// TwinCAT 3 PLC project IBF_Devices
// Title: IBF_Devices
// Company: Industrial Brains B.V.
// ProjectVersion: 0.0.0.0
// ProgramVersion: 3.1.4023.0
// CompilerDefines: InclSerialCom := 'true'
// libraries:
//   IBF_Utilities, * (Industrial Brains B.V.)
//   Tc2_Drive, * (Beckhoff Automation GmbH)
//   Tc2_EtherCAT, * (Beckhoff Automation GmbH)
//   Tc2_IoFunctions, * (Beckhoff Automation GmbH)
//   Tc2_Math, * (Beckhoff Automation GmbH)
//   Tc2_MC2, * (Beckhoff Automation GmbH)
//   Tc2_MC2_Drive, * (Beckhoff Automation GmbH)
//   Tc2_Standard, * (Beckhoff Automation GmbH)
//   Tc2_System, * (Beckhoff Automation GmbH)
//   Tc2_Utilities, * (Beckhoff Automation GmbH)
//   Tc3_Module, * (Beckhoff Automation GmbH)
//   VisuDialogs, * (System)
// project tree:
//   Axis/FunctionBlocks/Servo/ Fb_DevAxisDelta.TcPOU, Fb_DevAxis.TcPOU
//   / GlobalTextList.TcGTLO, PlcTask.TcTTO, Visualization Manager.TcVMO (not stored), VISU_TASK.TcTTO
//   GroupHandlers/ManualControlHandler/DataTypes/ UDT_DeviceID.TcDUT, UDT_HMI_ManualControl.TcDUT
//   GroupHandlers/ManualControlHandler/HMI/DeviceScreens/ VisuAnalogAxisControl.TcVIS, VisuAnalogOutControl.TcVIS, VisuAnlogInputControl.TcVIS, VisuAxisControl.TcVIS, VisuCylinderControl.TcVIS, VisuDigitalInputControl.TcVIS, VisuDigitalOutControl.TcVIS, VisuDoublePWMControl.TcVIS, VisuEncoderInput.TcVIS, VisuKL15XXControl.TcVIS, VisuKL5151Control.TcVIS, VisuPushbuttonLightControl.TcVIS, VisuPWMControl.TcVIS, VisuTwoVelocityAxisControl.TcVIS, VisuUndefinedControl.TcVIS, VisuValveControl.TcVIS
//   GroupHandlers/ManualControlHandler/HMI/ ManualControl.TcVIS
//   GVL/ GVL_Devices.TcGVL
//   _TESTS/ PRG_TEST_FB_DEVAXIS.TcPOU, PRG_TEST_FB_DEVVALVE.TcPOU, PRG_TEST_FB_MANUALCONTROLLER.TcPOU, PRG_TEST_GLOBAL.TcPOU, VISU_TEST.TcVIS, VISU_TEST_LOGIN.TcVIS
//   Actuators/Cylinder/DataTypes/ E_CylinderCmd.TcTLEO (not stored), E_ValveResetState.TcTLEO (not stored)
//   Actuators/Cylinder/DataTypes/ManualControls/ UDT_ManualValveControl.TcDUT (not stored)
//   Actuators/Cylinder/Functions/ Fb_DevCylWithFbk.TcPOU, FB_DevValve.TcPOU
//   Axis/DataTypes/ E_AxisCmd.TcTLEO (not stored), UDT_AxisData.TcDUT (not stored), UDT_AxVal.TcDUT (not stored), UDT_ManualAxisCtrl.TcDUT (not stored)
//   Axis/FunctionBlocks/Analog/ FB_DevAnalogAxis.TcPOU, ST_ManualAnalogAxisCtrl.TcDUT (not stored)
//   Axis/FunctionBlocks/ServoHybrid/ FB_DevBasicACAxis.TcPOU, FB_DevHybridAc.TcPOU
//   Axis/FunctionBlocks/TwoVelocityControl/DataTypes/ st_ManualDigitalMotorControl.TcDUT
//   Axis/FunctionBlocks/TwoVelocityControl/ FB_DevTwoVelocityAxis.TcPOU
//   Axis/Interface/ iTwoDirectionalMotor.TcIO, iTwoDirectionalMotorWithFast.TcIO (not stored)
//   BaseFunctions/ FB_DevBase.TcPOU, UDT_DevManualCtrl.TcDUT (not stored)
//   Buttons/Functions/ FB_DevHMIButton.TcPOU, FB_DevPushbuttonLight.TcPOU, FB_DevPushButton.TcPOU
//   CounterCards/FunctionBlocks/KL1512/ FB_DevKL1512.TcPOU (not stored)
//   CounterCards/FunctionBlocks/KL5151/ FB_DevKL5151.TcPOU
//   CounterCards/Interfaces/ iCounter.TcIO (not stored)
//   CounterCards/ st_ManualCounterControl.TcDUT (not stored)
//   DevTypes/ E_Devices.TcTLEO
//   Encoders/FunctionBlocks/ FB_EncoderBase.TcPOU, FB_EncoderInput.TcPOU
//   GroupHandlers/ManualControlHandler/ FB_ManualController.TcPOU
//   HardwareDiagnostics/ FB_ELModuleDiag.TcPOU (not stored)
//   Heaters/ FB_DevDoublePWM.TcPOU, FB_DevPWMGenerator.TcPOU
//   Lights/Functions/ Fb_DevLight.TcPOU
//   Outputs/AnalogOutputs/ FB_DevAnalogOutput.TcPOU, FB_DevAnalogOutputScaled.TcPOU
//   Outputs/DigitalOutputs/ FB_DevDigitalOutput.TcPOU
//   Sensors/AnalogInput/FunctionBlocks/ FB_DevAnalogInput.TcPOU, FB_DevAnalogInputScaled.TcPOU, FB_DevHDAnalogInAutoCalibrate.TcPOU, FB_DevAnalogInAutoCalibrate.TcPOU, FB_DevHDAnalogInputScaled.TcPOU, FB_DevHDAnalogInput.TcPOU
//   Sensors/DigitalSensor/FunctionBlocks/ Fb_DevDigitalInput.TcPOU, Fb_DevDigitalInputFunctions.TcPOU
//   Sensors/FootPedals/DataTypes/ E_FootpedalPos.TcTLEO (not stored)
//   Sensors/FootPedals/FunctionBlocks/ FB_EfkaEB301A_FootPedal.TcPOU
//   Sensors/ModuleSpecific/EL3556_Loadcell/ Fb_DevEL3356_LoadCell.TcPOU (not stored)
//   Version/ Global_Version.TcGVL
// real-time tasks:
//   TASK PlcTask: cycle T#10ms, priority 10, ADS port 350
//   TASK VISU_TASK: cycle T#200000us, priority 12, ADS port 351
// motion (NC):
//   TASK NC-Task 1 SAF: cycle T#2ms, priority 4, ADS port 501
//   TASK NC-Task 1 SVB: cycle T#10ms, priority 8, ADS port 511
//   AXIS Axis 1 (id 1)
//     OtherSettings: AllowMotionCmdToSlave=true
//     encoder EncType=1
//       SoftEndMinControl: Enable=true
//       SoftEndMaxControl: Enable=true, Range=1000
//     drive DrvType=5
//       Analog: TorqueSetpointScale=10, ScaleFactorActTorque=0.1
//       TimeComp: TaskDelayCycles=1
//     controller CtrType=1
//       CtrPara: PriorControlFactor=1
//         Observer: BandWidth=20
// variable links:
//   IBF_Devices Instance <-> NC-Task 1 SAF/Axes/Axis 1
//     PlcTask Inputs/PRG_TEST_FB_DEVAXIS.fbDevAxis.AxisRef.NcToPlc <-> Outputs/ToPlc
//     PlcTask Outputs/PRG_TEST_FB_DEVAXIS.fbDevAxis.AxisRef.PlcToNc <-> Inputs/FromPlc

CONFIGURATION IBF_Devices
    RESOURCE PLC ON TwinCAT3
        TASK PlcTask(INTERVAL := T#10ms, PRIORITY := 10);
        TASK VISU_TASK(INTERVAL := T#200000us, PRIORITY := 12);
        PROGRAM PRG_TEST_GLOBAL WITH PlcTask : PRG_TEST_GLOBAL;
        PROGRAM PRG_TEST_FB_DEVAXIS WITH PlcTask : PRG_TEST_FB_DEVAXIS;
        PROGRAM PRG_TEST_FB_DEVVALVE WITH PlcTask : PRG_TEST_FB_DEVVALVE;
        PROGRAM PRG_TEST_FB_MANUALCONTROLLER WITH PlcTask : PRG_TEST_FB_MANUALCONTROLLER;
        PROGRAM VisuElems_Visu_Prg WITH VISU_TASK : VisuElems.Visu_Prg;
    END_RESOURCE
END_CONFIGURATION

// ---- GroupHandlers/ManualControlHandler/DataTypes/UDT_DeviceID.TcDUT
TYPE UDT_DeviceID :
STRUCT
	sName			: STRING	; // device name
	sType			: STRING	; // Type of device [string for visu]
	pFunction		: POINTER TO FB_DevBase ; // Pointer to the device
END_STRUCT
END_TYPE

// ---- GroupHandlers/ManualControlHandler/DataTypes/UDT_HMI_ManualControl.TcDUT
TYPE UDT_HMI_ManualControl : // The link between HMI and FB
STRUCT
	refSelectedDevice	: REFERENCE TO FB_DevBase; // Reference to currently selected device
	nSelectedDevice		: UDINT; // Combo box index
	bReset 				: BOOL;
	bEnabled			: BOOL;	
	bBlocked			: BOOL;

	// References to all supported device types
	pDevValve			: POINTER TO FB_DevValve;
	pDevCylinder		: POINTER TO Fb_DevCylWithFbk; 
	pDevAxis			: POINTER TO Fb_DevAxis; 
	pDevPBL				: POINTER TO FB_DevPushbuttonLight;
	pDevDigitalInput	: POINTER TO Fb_DevDigitalInputFunctions;
	pDevAnalogInput		: POINTER TO FB_DevAnalogInput;
	pDevAnalogOut		: POINTER TO FB_DevAnalogOutput;
	pDevDigitalOut		: POINTER TO FB_DevDigitalOutput;
	pDevPWMController	: POINTER TO FB_DevPWMGenerator;
	pDevDoublePWM		: POINTER TO FB_DevDoublePWM;
	pDevEncoder			: POINTER TO FB_EncoderBase;
	pDevAnalogAxis		: POINTER TO FB_DevAnalogAxis;
	pDevTwoVelocityAxis	: POINTER TO FB_DevTwoVelocityAxis;
	pDevKL5151			: POINTER TO FB_DevKL5151;
	pDevKL1512			: POINTER TO FB_DevKL1512;
END_STRUCT
END_TYPE

// ---- Axis/FunctionBlocks/TwoVelocityControl/DataTypes/st_ManualDigitalMotorControl.TcDUT
TYPE st_ManualDigitalMotorControl : // commands from manual controller
STRUCT
	bManRunCW 		: BOOL ;
	bManRunCWFast	: BOOL ;
	bManRunCCw		: BOOL ;
	bManRunCCWFast	: BOOL ; 
END_STRUCT
END_TYPE

// ---- DevTypes/E_Devices.TcTLEO
{attribute 'qualified_only'}
{attribute 'strict'}
{attribute 'to_string'}
TYPE E_Devices :
(
	Undefined,
	Valve,
	Cylinder,
	Axis,
	PushButtonLight,
	DigitalSensor,
	AnalogSensor,
	DigitalOut,
	AnalogOut,
	PWMController,
	DoublePWMController,
	Encoder,
	AnalogAxis,
	TwoVelocityAxis,
	KL5151,
	KL1512
)INT;
END_TYPE

// ---- GVL/GVL_Devices.TcGVL
{attribute 'qualified_only'}
VAR_GLOBAL
	fbManualController : FB_ManualController;
END_VAR

// ---- Version/Global_Version.TcGVL
{attribute 'TcGenerated'}
{attribute 'no-analysis'}
{attribute 'linkalways'}
// This function has been automatically generated from the project information.
VAR_GLOBAL CONSTANT
	{attribute 'const_non_replaced'}
	stLibVersion_IBF_Devices : ST_LibVersion := (iMajor := 0, iMinor := 0, iBuild := 0, iRevision := 0, nFlags := 0, sVersion := '0.0.0.0');
END_VAR

// ---- Axis/Interface/iTwoDirectionalMotor.TcIO
INTERFACE iTwoDirectionalMotor // Two directional motor control

METHOD CmdRunCCW : BOOL
VAR_INPUT
END_VAR
END_METHOD

METHOD CmdRunCW : BOOL
VAR_INPUT
END_VAR
END_METHOD

METHOD Init : BOOL
VAR_INPUT
	// Message location data
	nId				: UINT ; // Identification number of object
	nParentId		: UDINT ; // Id of higher level If aplicable (0 = no parent)
END_VAR
END_METHOD

END_INTERFACE

// ---- _TESTS/PRG_TEST_GLOBAL.TcPOU
PROGRAM INTERNAL PRG_TEST_GLOBAL // A place to call global function blocks (singletons) that can be used by all tests

Sys_Variables.fbSystemVariables();
GVL_Utilities.fbFaultHandler();

END_PROGRAM

// ---- _TESTS/PRG_TEST_FB_DEVAXIS.TcPOU
PROGRAM INTERNAL PRG_TEST_FB_DEVAXIS
VAR
	bEnableTests : BOOL;
	
	fbDevAxis : Fb_DevAxis;
	
	// Setpoints
	fVelocity : LREAL := 100;
	fPosition : LREAL := 500; // NOTE: software limit switch is at 1000 (/Axes/Axis 1/Enc/ Parameters)

	// Public commands
	bInit : BOOL;
	bCmdHalt : BOOL;
	bCmdHold : BOOL;
	bCmdHome : BOOL;
	bCmdReset : BOOL;
	bCmdMoveAbs : BOOL;
END_VAR

IF bEnableTests THEN
	fbDevAxis();
	
	IF bInit THEN
		bInit R= fbDevAxis.Init(
			nId					:= 1, 
			nParentId			:= 0, 
			bIcfCmdVelocityRpm	:= FALSE, 
			bIcfEnableForward	:= TRUE, 
			bIcfEnableReverse	:= TRUE, 
			bIcfAlwaysEnable	:= FALSE, 
			bIcfModuloAxis		:= FALSE, 
			bIcfSTOPresent		:= TRUE, 
			bIcfNCHomeSensor	:= FALSE, 
			mcHomingMode		:= MC_HomingMode.MC_DefaultHoming, 
			fSafeOverride		:= 20, 
			nEncTurnoverVal		:= 0,
			tEnableDelay		:= T#0S, 
			tDisabledelay		:= T#200MS
		);
	END_IF
		
	// Trigger commands
	IF bCmdHalt THEN bCmdHalt R= fbDevAxis.CmdHalt(fDeceleration := 1000, MC_BufferMode.MC_Aborting); END_IF
	IF bCmdHold THEN bCmdHold R= fbDevAxis.CmdHold(); END_IF
	IF bCmdHome THEN bCmdHome R= fbDevAxis.CmdHome(); END_IF
	IF bCmdReset THEN bCmdReset R= fbDevAxis.CmdReset(); END_IF
	IF bCmdMoveAbs THEN bCmdMoveAbs R= fbDevAxis.CmdMoveAbs(fPosition := fPosition, fVelocity := fVelocity, MC_BufferMode.MC_Aborting); END_IF
END_IF

END_PROGRAM

// ---- Axis/FunctionBlocks/Servo/Fb_DevAxis.TcPOU
{attribute 'reflection'}
FUNCTION_BLOCK PUBLIC Fb_DevAxis EXTENDS FB_DevBase
VAR_INPUT
	// ===== General Function input =====
		fCmdAcc			: LREAL := 15000;
		fCmdDec			: LREAL := 15000; 
	// ===== Master Axis =====
		refMasterAxis	: REFERENCE TO AXIS_REF ; // Master axis reference (if applicable)
		bReverseSlave	: BOOL 	:= FALSE; // Reverse slave axis relative to master
		fCmdGearRatio	: LREAL := 1 ; // Gear ratio Master/Slave (1/Ratio) 
	// Manual control reference
		stManualCtrl	: UDT_ManualAxisCtrl ;
END_VAR
VAR_OUTPUT
	// ====== State indications =======
		bHomed			: BOOL 	:= FALSE; 
		bError 			: BOOL 	:= FALSE;
		bStopped		: BOOL 	:= FALSE;
		bResetDone		: BOOL 	:= FALSE;
		bGearedAsSlave	: BOOL 	:= FALSE;
		bVelocityLimited: BOOL 	:= FALSE;  
		bIdle			: BOOL 	:= FALSE;
		fVelocity		: LREAL	:= 0	; // Axis velocity [rpm or units/sec] depending on config
		fActPosition	: LREAL := 0	; // Axis actual position [Units] depending on config	
		bReInTargetPos	: BOOL 	:= false; // rising edge axis is in position
	// ====== axis reference ======
		AxisRef			: AXIS_REF	; // Axis reference to hardware 
	// ====== Axis Settings ======
		fMaxVelo		: LREAL := 0 ; // Axis Maximum velocity
		fMaxAcc			: LREAL := 0 ; // Axis Maximum cceleration
		fMaxDec			: LREAL := 0 ; // axis Maxium deceleration 
	
//		fSafeVeloLimit	: LREAL	:= 200; // Safe velocity limit 
		tEnableDelay	: TIME 	:= T#0MS	;
		tDisableDelay	: TIME 	:= T#500MS  ;
	// ==== Axis data ====
		fEncoderTurnoverValue	: LREAL ;   
		
END_VAR
VAR // Axis configuration 
	// ===== HW Config Bits =====
		bIcfCmdVelocityRpm	: BOOL ; // input speeds in Rpm
		bIcfEnableForward 	: BOOL ; // Enable forward motion
 		bIcfEnableReverse	: BOOL ; // Enable reverse motion
		bIcfAlwaysEnable	: BOOL ; // 1 = Axis always enabled, 0 = Axis disabled at Idle 
		bIcfModuloAxis		: BOOL := FALSE ; // Show axis position as modulo
		bIcfSTOPresent		: BOOL := FALSE ; // Axis Safe torque off is present
		bIcfNCHomeSensor	: BOOL := FALSE ; // Homing sensor is inverted (NC)	
	// Command Modes
		mcHomingMode 		: MC_HomingMode := MC_direct ; // Homing Mode ( MC_DefaultHoming, MC_Direct, MC_ForceCallibration, MC_ResetCallibration)
	// Values from system
		McReadSysVelo		: MC_ReadParameter		; // Read Acceleration parameter from drive 
		McReadSysAcc		: MC_ReadParameter		; // Read Acceleration parameter from drive 
		McReadSysDec		: MC_ReadParameter		; // Read Acceleration parameter from drive 
END_VAR
VAR	// ====== Axis enable =====
		bCmdEnableAxis 		: BOOL 	:= FALSE; // Command to enable the axis (External)
		bInternalEnable		: BOOL 	:= FALSE; // internal enable command (turns off after set time, and on at new motion command
		bAxisIsEnabled		: BOOL 	:= false; // Axis is enabled and ready for commands
		bDelayedEnable		: BOOL 	:= false; // Delayed enable signal for motion commands
		TonMotionEnable		: TON 			; // Timer on for motion command enable
		TofIntAxisEnable	: TOF  			; // Timer off for internal axis enable 
		bSTOOK				: BOOL 	:= FALSE; // Axis safet torque off is ok
		tonSTOOK			: TON	; // Safe torque off ok timer
	// Parameter read status 
		Cmd_EnDriveParRead	: BOOL 			; // Enable parameter read 
	// ===== Physical Homing signal =====
		IAxisHome 	AT %I* 	: BOOL 			; // Axis homing sensor from PLC (if MC_DefaultHoming is used)
		IAxisSTOOK	AT %I* 	: BOOL 			; // Axis STO is ok
END_VAR
VAR	// =============== Motion status functions ================
	// =============== Motion function blocks =================
		fbMcPower 			: MC_Power		;		// FB for enable and override
		fbMcReset 			: MC_Reset		;		// FB to reset axis
		fbSoeReset			: FB_SoEReset	; 		// FB to reset axis hardware
		fbMcHome			: MC_Home		;		// Fb to home Axis
		fbHomeResetCalibrationFlag:MC_Home;			// Fb to clear calibration (homed) bit
		bResetCalibrationFlag : BOOL := FALSE; // When TRUE, the calibration bit (homing OK) will be reset. Set to TRUE on homing faults.
		fbMcStop 			: MC_Stop		;		// FB to stop axis
		fbMcHalt			: MC_Halt		;		// FB to halt axis
		fbMcJog				: MC_Jog		;		// FB to Jog axis
		fbMcMoveVelocity	: MC_MoveVelocity;		// FB to move with specified velocity until Next command is given
		fbMcGearInSlave		: MC_GearIn		;		// FB to gear axis to master 
		fbMcGearInDyn		: MC_GearInDyn	;		// FB to gear axis dynamicly to master
		fbMcGearOutSlave	: MC_GearOut	;		// FB to decouple gearing
		fbMcSetPosition		: MC_SetPosition;		// FB to Set axis position
//		fbMcWriteParameter	: MC_WriteParameterPersistent ; // FB to write parameters in persistend data

	(* PtoP Motion move commands are in arrays so multiple commands can be stacked *) 
		fbMCMoveRelative	: ARRAY [0..1] OF MC_MoveRelative	;		// FB to move relative
		fbMcMoveAbsolute	: ARRAY [0..1] OF MC_MoveAbsolute	;		// FB to move axis (velocity movement)
		fbMcMoveModulo		: ARRAY [0..1] OF MC_MoveModulo		;		// FB to move axis to modulo position
	// ===== Safe commands =====
		bCmdSafeStop		: BOOL ;
		bCmdSafeSpeed		: BOOL ; 
	// ===== Function execute triggers =====
		bExec_Reset					: BOOL := FALSE; // Execute reset
		bExec_Halt					: BOOL := FALSE; // Execute hold
		bExec_Home					: BOOL := FALSE; // Execute Home
		bExec_JogPositive			: BOOL := FALSE; // Execute Jog in positive direction
		bExec_JogNegative			: BOOL := FALSE; // Execute Jog in negative direction
		bExec_MoveVelocity			: BOOL := FALSE; // Execute move velocity
		bExec_MoveVelocityDynamic	: BOOL := FALSE; // Execute move velocity
		bExec_GearAsSlave			: BOOL := FALSE; // Execute gear as slave
		bExec_GearSlaveDyn			: BOOL := FALSE; // Execute gear slave dynamic
		bExec_GearOutSlave			: BOOL := FALSE; // Execute gear out slave
		bExec_SetPosition			: BOOL := FALSE; // execute set position
		
	(* PtoP Motion move commands are in arrays so multiple commands can be stacked *) 
		arExec_MoveRelative	: ARRAY [0..1] OF BOOL ; // Execute move relative
		arExec_MoveAbs		: ARRAY [0..1] OF BOOL ; // Execute move absolute reverse
		arExec_MoveModulo	: ARRAY [0..1] OF BOOL ; // Execute move modulo

		tonResetDone		: TON := (PT := T#300MS) ;

	// ===== Move ristrictions ======
		bCmdLimitVelocity 	: BOOL := FALSE			; // velocity limiting is active 
		fCmdVelocityLimit	: LREAL:= 100			; // Maximum velocity limit when velocity limiting is active  
		fSafeOverride		: LREAL:= 10 			; // [%] Safe velocity override  
		
	// ===== Internal variables =======
		fAcceleration		: LREAL := 0 ; // Acceleration used for functions 
		fDeceleration		: LREAL := 0 ; // Deceleration used for functions
		fLastCommandPosition: LREAL := 0 ; // Last given position command
		fLastCommandVelocity: LREAL := 0 ; // Last given Velocity command

	// Register command changes to make sure CmdMoveAbs is triggered
	{warning 'TODO: this is a workaround for a generic software design issue of DevAxis (needs state machine)'}
	bResetCmdMoveAbs : BOOL := TRUE;
		
END_VAR
VAR
	// ===== Loop variables =====
		i : DINT := 0 ; // For loop increment
	// ===== check variable ======
		rtrigInPosition	: R_TRIG ; // in position trigger
	// ===== Par write timer ===== 
END_VAR
VAR // Parameters 
	ParHomeOffset		: Udt_Parameter := (fValue := 0, fFactory := 0, bTeachable := FALSE)	; // Home position offset
END_VAR

// Call base function
SUPER^();

// ==== Check if axis is initiated =====
IF NOT bInitOk THEN 
	RETURN ; 
END_IF
// ===== Execute safe functions =====
	ExecSafeFunctions(); 
	
// ==== Execute organizational functions =====
	CallOrganizationFunctions();
// ==== execute motion functions =====
	CallMotionFunctions();

// ==== reset calibration ("homed") flag =====
fbHomeResetCalibrationFlag(
  Execute:=bResetCalibrationFlag,
  HomingMode:=MC_ResetCalibration,
  Axis:=AxisRef
);
bResetCalibrationFlag R= fbHomeResetCalibrationFlag.Done;


IF bHomed AND (NOT AxisRef.NcToPlc.StateDWord.1) // Check if drive is still homed
THEN 
	{warning 'TODO: Skip homing check if the drive is not connected (e.g., during automated tests of an axis with disabled hardware)'}
	bHomed := FALSE;
	IF NOT bManual THEN // Ignore homing error when in manual mode
		bError					:= TRUE							;
		stFault.Active 			:= TRUE 						;
		stFault.Description		:= 'Axis no longer homed';
		stFault.FaultType		:= E_FaultTypes.FF				;	
	END_IF
END_IF

METHOD PRIVATE CallMotionFunctions : BOOL
VAR_INPUT
END_VAR
// ===== block all other commands if axis is coupled =====
	IF NOT AxisRef.Status.Coupled THEN 
	// ===== Homing functions =====
		ExecHome		(); 
	
	// ===== Motion standstil commands =====
		ExecHalt		();
	
	// ===== Motion move functions
		ExecJog			();
		ExecMoveAbsolute();
		ExecMoveRelative();
		ExecMoveModulo	();
		ExecMoveVelocity();
	END_IF
	
// ===== Execute gearing functions =====
 IF __ISVALIDREF (refMasterAxis) THEN 
	ExecGearOut		();
	ExecGearIn		();
	ExecGearDynamic	();
 END_IF
	
// ====== reset velocity lmiting =====
	bVelocityLimited	:= bCmdLimitVelocity ;	
	bCmdLimitVelocity 	:= FALSE ; 

// ====== Reset acceleration deceleration values ======
	fAcceleration	:= fCmdAcc;
	fDeceleration	:= fCmdDec;
END_METHOD

METHOD PRIVATE CallOrganizationFunctions : BOOL
VAR_INPUT
END_VAR
// ==== execute organizational functions =====
	ExecReadStatus		(); 
	ExecEnable			();
	ExecReset			();
//	ExecWriteParameter	();
	ExecSetPosition		();
END_METHOD

METHOD PUBLIC CmdGearDynamic : BOOL // Set axis to geared, activates with variable gear ratio until geared out or stopped (if method is no longer called then gear ratio is locked to last value)
VAR_INPUT
	fGearRatio	:	LREAL	:= 1	; // Slave Axis gearing ratio (Master = 1/ fGearRatio = Slave)	
END_VAR
// check if master is present
	IF NOT __ISVALIDREF (refMasterAxis) THEN 
		bError					:= TRUE							;
		stFault.Active 			:= TRUE 						;
		stFault.Description		:= CONCAT('Axis master not found ', UDINT_TO_STRING(fbMcHalt.ErrorID));
		stFault.FaultType		:= E_FaultTypes.FF				;
	END_IF

// check if error is active
	IF bError THEN
		stFault.Active 			:= TRUE 						;
		stFault.Description		:= 'Call to CmdGearDynamic while axis has an error';
		stFault.FaultType		:= E_FaultTypes.CF				;	
		RETURN;
	END_IF

// set blocked command if halt is active 
	bBlockedCommand 		:= fbMcHalt.Active ;


// check if command buffer is empty 
	IF AxisRef.Status.CmdBuffered THEN 
		RETURN ;
	END_IF 

// Set command to true 
	bExec_GearSlaveDyn 	:= TRUE ;
	bInternalEnable		:= TRUE ;

// copy parameters
	fCmdGearRatio 		:= fGearRatio ;

// Reset CmdMoveAbs
bResetCmdMoveAbs := TRUE;

// Set feedback output 
	CmdGearDynamic 		:= bGearedAsSlave ;
END_METHOD

METHOD PUBLIC CmdGearIn : BOOL // Set axis to geared, activates with constant gear ratio until geared out or stopped
VAR_INPUT
	fGearRatio	:	LREAL	:= 1	; // Slave Axis gearing ratio (Master = 1/ fGearRatio = Slave)	
END_VAR
// Check if master is present
	IF NOT __ISVALIDREF (refMasterAxis) THEN 
		bError					:= TRUE							;
		stFault.Active 			:= TRUE 						;
		stFault.Description		:= CONCAT('Axis master not found ', UDINT_TO_STRING(fbMcHalt.ErrorID));
		stFault.FaultType		:= E_FaultTypes.FF				;
	END_IF

// check if error is active
	IF bError THEN
		stFault.Active 			:= TRUE 						;
		stFault.Description		:= 'Call to CmdGearIn while axis has an error';
		stFault.FaultType		:= E_FaultTypes.CF				;	
		RETURN;
	END_IF

// set blocked command if halt is active 
	bBlockedCommand := fbMcHalt.Active ;

// check if command buffer is empty 
	IF AxisRef.Status.CmdBuffered THEN 
		RETURN ;
	END_IF 
	
// Set command to true 
	bExec_GearAsSlave 	:= TRUE ;
	bInternalEnable		:= TRUE ;

// copy parameters
	fCmdGearRatio 				:= fGearRatio ;

// Reset CmdMoveAbs
bResetCmdMoveAbs := TRUE;

// Set feedback output 
	CmdGearIn := bGearedAsSlave ;
END_METHOD

METHOD CmdGearOut : BOOL
VAR_INPUT
END_VAR
// Check if master is present
	IF NOT __ISVALIDREF (refMasterAxis) THEN 
		bError					:= TRUE							;
		stFault.Active 			:= TRUE 						;
		stFault.Description		:= CONCAT('Axis master not found ', UDINT_TO_STRING(fbMcHalt.ErrorID));
		stFault.FaultType		:= E_FaultTypes.FF				;
	END_IF

// check if error is active
	IF bError THEN
		stFault.Active 			:= TRUE 						;
		stFault.Description		:= 'Call to CmdGearOut while axis has an error';
		stFault.FaultType		:= E_FaultTypes.CF				;	
		RETURN;
	END_IF

// set blocked command if halt is active 
bBlockedCommand := fbMcHalt.Active ;

// Set command to true
bExec_GearOutSlave 	:= TRUE ;
bExec_GearAsSlave	:= FALSE;
bExec_GearSlaveDyn 	:= FALSE;

// Reset CmdMoveAbs
bResetCmdMoveAbs := TRUE;

// Set feedback Output
CmdGearOut := fbMcGearOutSlave.Done;
END_METHOD

METHOD PUBLIC CmdHalt : BOOL
VAR_INPUT
	fDeceleration 	: LREAL := 0 ; // command deceleration
	mcBuffermode	: MC_BufferMode ; // Buffermode defines how the previous command is executed.
END_VAR
// Set command to true 
bExec_Halt 		:= TRUE ;
bInternalEnable	:= TRUE ;

// copy parameters
fbMcHalt.Deceleration	:= fDeceleration;
fbMcHalt.BufferMode		:= mcBuffermode	;

// Reset CmdMoveAbs
bResetCmdMoveAbs := TRUE;

// Set feedback output 
CmdHalt := fbMchalt.Active OR fbMcHalt.Done ;
END_METHOD

METHOD PUBLIC CmdHold : BOOL
VAR_INPUT
END_VAR
// Set command to true 
bExec_Halt 		:= TRUE ;
bInternalEnable	:= TRUE ;

// copy parameters
fbMcHalt.Deceleration	:= 0;
fbMcHalt.BufferMode		:= 0;
	
// Reset CmdMoveAbs
bResetCmdMoveAbs := TRUE;

// Set feedback output 
CmdHold := fbMchalt.Active OR fbMcHalt.Done ;
END_METHOD

METHOD PUBLIC CmdHome : BOOL // start axis homing procedure
// set blocked command if halt is active 
bBlockedCommand := fbMcHalt.Active ;

// check if error is active
	IF bError THEN
		stFault.Active 			:= TRUE 						;
		stFault.Description		:= 'Call to CmdHome while axis has an error';
		stFault.FaultType		:= E_FaultTypes.CF				;	
		RETURN;
	END_IF

// Enable drive 
bExec_Home 		:= NOT bResetCalibrationFlag; 
bInternalEnable	:= TRUE ;

// copy parameters
fbMcHome.Position 	:= ParHomeOffset.fValue;

// Reset CmdMoveAbs
bResetCmdMoveAbs := TRUE;

// Set feedback output
CmdHome := fbMcHome.Done ;
END_METHOD

METHOD PUBLIC CmdJog : BOOL // Jog axis with variable speed. jog stops as soon as the command is false
VAR_INPUT
	fVelocity		: LREAL 	; // jog velocity can be adjusted as long as the command is active
	fPos			: LREAL 	; // Jog position or step size (if aplicable)
	bJogNegative 	: BOOL 		:= FALSE ; // jog in negative direction
	eJogmode		: E_JogMode := E_JogMode.MC_JOGMODE_CONTINOUS ; // jogmode [default MC_JOGMODE_CONTINOUS] 
END_VAR
// set blocked command if halt is active 
bBlockedCommand := fbMcHalt.Active ;

// check if error is active
	IF bError THEN
		stFault.Active 			:= TRUE 						;
		stFault.Description		:= 'Call to CmdJog while axis has an error';
		stFault.FaultType		:= E_FaultTypes.CF				;	
		RETURN;
	END_IF

// Velocity conversion from RPM to deg/sec
	IF bIcfCmdVelocityRpm THEN 
		fVelocity := Rpm_To_DegS(fVelocity);
	END_IF

// Set command to true
	IF fbMcJog.Velocity = fVelocity THEN // If command velocity changes, then set exec to false for one cycle to trigger new velocity so the jog follows the set velocity
		bExec_JogPositive	:= NOT bJogNegative ;
		bExec_JogNegative 	:= bJogNegative ;
	END_IF
	bInternalEnable			:= TRUE ;

// copy parameters
	fbMcJog.Velocity	:= fVelocity 	;
	fbmcjog.Mode		:= eJogmode		;
	fbMcJog.Position	:= fPos			;

// Reset CmdMoveAbs
bResetCmdMoveAbs := TRUE;

// Set feedback output 
	CmdJog := fbMcJog.Active ;
END_METHOD

METHOD PUBLIC CmdKeepEnabled : BOOL
VAR_INPUT
END_VAR
// Keep internal enable on while command is active
bInternalEnable			:= TRUE ;
END_METHOD

METHOD PUBLIC CmdLimitVelocity : BOOL // limit axis maximum velocity, stays active as long as command is called. 
VAR_INPUT
	fVelocityLimit	: LREAL ; // velocity Maximum limit
END_VAR
// set blocked command if halt is active 
bBlockedCommand := fbMcHalt.Active ;

// Set velocity limiting command 
bCmdLimitVelocity S= TRUE;
	
// Set velocity maximum value 
fCmdVelocityLimit := fVelocityLimit ; 

// set feedback 
CmdLimitVelocity := bVelocityLimited ;
END_METHOD

METHOD PUBLIC CmdManual : BOOL
VAR
	eJogmode		: E_JogMode := E_JogMode.MC_JOGMODE_CONTINOUS ; // jogging mode 
END_VAR
// set blocked command if halt is active 
bBlockedCommand := fbMcHalt.Active ;

// Enable axis for manual control
bCmdManual := TRUE ;

// set jog mode 
IF stManualCtrl.bCmdInching THEN 
	eJogmode := E_JogMode.MC_JOGMODE_INCHING ;
END_IF

// execute motion commands
IF stManualCtrl.bCmdJogForward OR stManualCtrl.bCmdJogReverse THEN 
	CmdJog (fVelocity := stManualCtrl.fVelocity, 
			fPos := stManualCtrl.fDistance, 
			bJogNegative := stManualCtrl.bCmdJogReverse, 
			eJogmode := eJogmode);
ELSIF stManualCtrl.bCmdToPos THEN 
	CmdMoveAbs( fPosition := stManualCtrl.fPosition, 
				fVelocity := stManualCtrl.fVelocity, 
				mcBuffermode := MC_BufferMode.MC_Aborting);
ELSIF stManualCtrl.bCmdHome THEN 
	CmdHome();
ELSE 
	CmdHalt( 	fDeceleration := fMaxDec * 0.9, 
				mcBuffermode := MC_BufferMode.MC_Aborting) ; 
END_IF
END_METHOD

METHOD PUBLIC CmdMoveAbs : BOOL // Move absolute command
VAR_INPUT
	fPosition	:	LREAL 	; // target position
	fVelocity	: 	LREAL 	; // Maximum velocity [units/sec]
	mcBuffermode: 	MC_BufferMode ; // Buffermode defines how the previous command is executed.
END_VAR
VAR
	bNewCommandReceived : BOOL ;
END_VAR
IF (NOT AxisRef.NcToPlc.StateDWord.1) THEN
	bError					:= TRUE							;
	stFault.Active 			:= TRUE 						;
	stFault.Description		:= 'Unable to execute move command, axis not homed';
	stFault.FaultType		:= E_FaultTypes.FF				;	
	RETURN;
END_IF

// check if error is active
	IF bError THEN
		stFault.Active 			:= TRUE 						;
		stFault.Description		:= 'Call to CmdMoveAbs while axis has an error';
		stFault.FaultType		:= E_FaultTypes.CF				;	
		RETURN;
	END_IF

// set blocked command if halt is active 
bBlockedCommand := fbMcHalt.Active ;

// Velocity conversion from RPM to deg/sec
	IF bIcfCmdVelocityRpm THEN 
		fVelocity := Rpm_To_DegS(fVelocity);
	END_IF

// Determine if a new command is geven or previous command is repeated
bNewCommandReceived := bResetCmdMoveAbs
			OR (fPosition <> fLastCommandPosition) 
			OR (fVelocity <> fLastCommandVelocity)
;
bResetCmdMoveAbs := FALSE;

	
// Determine function for command stacking
IF mcBuffermode = MC_Aborting OR NOT AxisRef.Status.CmdBuffered THEN 
	IF NOT fbMcMoveAbsolute[0].Busy THEN
		arExec_MoveAbs[0] 				S= bNewCommandReceived ;
		fbMcMoveAbsolute[0].Position 	:= fPosition ;
		fbMcMoveAbsolute[0].Velocity 	:= fVelocity ; 
		fbMcMoveAbsolute[0].BufferMode 	:= mcBuffermode ;
	ELSE
		arExec_MoveAbs[1] 				S= bNewCommandReceived ;
		fbMcMoveAbsolute[1].Position 	:= fPosition ;
		fbMcMoveAbsolute[1].Velocity 	:= fVelocity ; 
		fbMcMoveAbsolute[1].BufferMode 	:= mcBuffermode ;
	END_IF
	fLastCommandPosition := fPosition;
	fLastCommandVelocity := fVelocity;
END_IF
	
bInternalEnable	:= TRUE ;

// set feedback
IF fbMcMoveAbsolute[0].Busy THEN 
	CmdMoveAbs :=	fbMcMoveAbsolute[0].Active ;
ELSE 
	CmdMoveAbs :=	fbMcMoveAbsolute[1].Active ;
END_IF
END_METHOD

METHOD PUBLIC CmdMoveModulo : BOOL // Move to a modulo position
VAR_INPUT
	fPosition	:	LREAL 	; // target position
	fVelocity	: 	LREAL 	; // Maximum velocity [units/sec]
	mcDirection : 	MC_Direction := MC_Direction.MC_Positive_Direction ; // Direction of movement mc_direction [ deafult mc_positive_direction]
	mcBuffermode: 	MC_BufferMode ; // Buffermode defines how the previous command is executed.
END_VAR
// set blocked command if halt is active 
bBlockedCommand := fbMcHalt.Active ;


// check if error is active
	IF bError THEN
		stFault.Active 			:= TRUE 						;
		stFault.Description		:= 'Call to CmdMoveModulo while axis has an error';
		stFault.FaultType		:= E_FaultTypes.CF				;	
		RETURN;
	END_IF

// Velocity conversion from RPM to deg/sec
	IF bIcfCmdVelocityRpm THEN 
		fVelocity := Rpm_To_DegS(fVelocity);
	END_IF

// Determine function for command stacking
IF NOT AxisRef.Status.CmdBuffered OR mcBuffermode <> MC_Aborting THEN 
	IF fbMcMoveModulo[0].Busy THEN 
		arExec_MoveModulo[1] 		:= (fPosition <> fbMcMoveModulo[0].Position OR fVelocity <> fbMcMoveModulo[0].Velocity)	;
		fbMcMoveModulo[1].Velocity 	:= fVelocity 	;
		fbMcMoveModulo[1].Position 	:= fPosition 	;
		fbMcMoveModulo[1].Direction	:= mcDirection	;
		fbMcMoveModulo[1].BufferMode:= mcBuffermode ;
	ELSE    
		arExec_MoveModulo[0] 		:= (fPosition <> fbMcMoveModulo[1].Position OR fVelocity <> fbMcMoveModulo[1].Velocity) ;
		fbMcMoveModulo[0].Velocity 	:= fVelocity 	;
		fbMcMoveModulo[0].Position 	:= fPosition 	;
		fbMcMoveModulo[0].Direction	:= mcDirection	;
		fbMcMoveModulo[0].BufferMode:= mcBuffermode ;
	END_IF
END_IF 
	
bInternalEnable	:= TRUE ;

// Reset CmdMoveAbs
bResetCmdMoveAbs := TRUE;

// set feedback
IF arExec_MoveModulo[1] OR fbMcMoveModulo[1].Busy THEN 
	CmdMoveModulo :=	fbMcMoveModulo[1].Active OR fbMcMoveModulo[1].Done;
ELSE
	CmdMoveModulo :=	fbMcMoveModulo[0].Active OR fbMcMoveModulo[0].Done ;
END_IF
END_METHOD

METHOD CmdMoveRelative : BOOL // move relative command 
VAR_INPUT
	fDistance	:	LREAL 	; // target position
	fVelocity	: 	LREAL 	; // Maximum velocity [units/sec]
	mcBuffermode: 	MC_BufferMode ; // Buffermode defines how the previous command is executed.
END_VAR
// set blocked command if halt is active 
bBlockedCommand := fbMcHalt.Active ;

// check if error is active
	IF bError THEN
		stFault.Active 			:= TRUE 						;
		stFault.Description		:= 'Call to CmdMoveRelative while axis has an error';
		stFault.FaultType		:= E_FaultTypes.CF				;	
		RETURN;
	END_IF

// Velocity conversion from RPM to deg/sec
	IF bIcfCmdVelocityRpm THEN 
		fVelocity := Rpm_To_DegS(fVelocity);
	END_IF

// Determine function for command stacking
IF NOT AxisRef.Status.CmdBuffered OR mcBuffermode <> MC_Aborting THEN 
	IF fbMCMoveRelative[0].Active THEN 
		arExec_MoveRelative[1] := (fDistance <> fbMCMoveRelative[0].Distance OR fVelocity <> fbMCMoveRelative[0].Velocity) ;
		fbMCMoveRelative[1].Velocity	:= fVelocity 	;
		fbMCMoveRelative[1].Distance	:= fDistance	;
		fbMCMoveRelative[1].BufferMode	:= mcBuffermode	;
	ELSE 
		arExec_MoveRelative[0] := (fDistance <> fbMCMoveRelative[1].Distance OR fVelocity <> fbMCMoveRelative[1].Velocity) ;
		fbMCMoveRelative[0].Velocity	:= fVelocity 	;
		fbMCMoveRelative[0].Distance	:= fDistance	;
		fbMCMoveRelative[0].BufferMode	:= mcBuffermode	;
	END_IF
END_IF
bInternalEnable	:= TRUE ;

// Reset CmdMoveAbs
bResetCmdMoveAbs := TRUE;

// set feedback
IF arExec_MoveRelative[1] OR fbMCMoveRelative[1].Busy THEN 
	CmdMoveRelative :=	fbMCMoveRelative[1].Active ;
ELSE
	CmdMoveRelative :=	fbMCMoveRelative[0].Active ;
END_IF
END_METHOD

METHOD PUBLIC CmdMoveVelocity : BOOL // Move with set velocity until stopped
VAR_INPUT
	fVelocity	: 	LREAL 	; // Maximum velocity [units/sec]
	mcDirection : 	MC_Direction := MC_Direction.MC_Positive_Direction ; // Direction of movement mc_direction [ deafult mc_positive_direction]
	mcBuffermode: 	MC_BufferMode ; // Buffermode defines how the previous command is executed.
END_VAR
// set blocked command if halt is active 
bBlockedCommand := fbMcHalt.Active ;

// check if error is active
	IF bError THEN
		stFault.Active 			:= TRUE 						;
		stFault.Description		:= 'Call to CmdMoveVelocity while axis has an error';
		stFault.FaultType		:= E_FaultTypes.CF				;	
		RETURN;
	END_IF

// Velocity conversion from RPM to deg/sec
	IF bIcfCmdVelocityRpm THEN 
		fVelocity := Rpm_To_DegS(fVelocity);
	END_IF

// Set command to true 
	IF NOT AxisRef.Status.CmdBuffered OR mcBuffermode <> MC_Aborting THEN 
		bExec_MoveVelocity 	:= TRUE ;
		bInternalEnable		:= TRUE ;
	END_IF
	
// copy parameters
	fbMcMoveVelocity.Velocity	:= fVelocity 	;
	fbMcMoveVelocity.Direction 	:= mcDirection	;
	fbMcMoveVelocity.BufferMode	:= mcBuffermode	;

// Reset CmdMoveAbs
bResetCmdMoveAbs := TRUE;

// Set feedback output 
	CmdMoveVelocity := fbMcMoveVelocity.Active ;
END_METHOD

METHOD PUBLIC CmdMoveVelocityDynamic : BOOL // Move with set velocity until stopped
VAR_INPUT
	fVelocity	: 	LREAL 	; // Maximum velocity [units/sec]
	mcDirection : 	MC_Direction := MC_Direction.MC_Positive_Direction ; // Direction of movement mc_direction [ deafult mc_positive_direction]
	mcBuffermode: 	MC_BufferMode ; // Buffermode defines how the previous command is executed.
END_VAR
VAR
	xbNewCmdVelocity : BOOL ; // a new command velocity has been detected
END_VAR
// set blocked command if halt is active 
bBlockedCommand := fbMcHalt.Active ;

// check if error is active
	IF bError THEN
		stFault.Active 			:= TRUE 						;
		stFault.Description		:= 'Call to CmdMoveVelocityDynamic while axis has an error';
		stFault.FaultType		:= E_FaultTypes.CF				;	
		RETURN;
	END_IF

// Velocity conversion from RPM to deg/sec
	IF bIcfCmdVelocityRpm THEN 
		fVelocity := Rpm_To_DegS(fVelocity);
	END_IF

// check for command velocity changes
	IF fVelocity > 0 THEN 	
		xbNewCmdVelocity := fbMcMoveVelocity.Velocity <> fVelocity OR NOT fbMcMoveVelocity.Active ;
	ELSE
		bExec_Halt := TRUE;
		fbMcHalt.Deceleration	:= fCmdDec;
		fbMcHalt.BufferMode		:= mcBuffermode	;
	END_IF
	
// Set command to true for one cycle
	IF (NOT AxisRef.Status.CmdBuffered OR mcBuffermode <> MC_Aborting) AND fVelocity > 0 THEN 
		bExec_MoveVelocityDynamic 	:= xbNewCmdVelocity;
		bInternalEnable				:= TRUE ;
	END_IF
	
// copy parameters
	fbMcMoveVelocity.Velocity	:= fVelocity 	;
	fbMcMoveVelocity.Direction 	:= mcDirection	;
	fbMcMoveVelocity.BufferMode	:= mcBuffermode	;

// Reset CmdMoveAbs
bResetCmdMoveAbs := TRUE;
	

// Set feedback output
	CmdMoveVelocityDynamic := fbMcMoveVelocity.Active ;
END_METHOD

METHOD PUBLIC CmdOverwriteAcc : BOOL // temporarilly overwrite deceleration values
VAR_INPUT	
	fValue	: LREAL ; // Overwrite value 
END_VAR
fAcceleration := fValue ;

CmdOverwriteAcc := TRUE ;
END_METHOD

METHOD PUBLIC CmdOverwriteDec : BOOL // Temporarilly overwrite deceleration values
VAR_INPUT
	fValue	: LREAL ; // Overwrite value 
END_VAR
fDeceleration := fValue ;

CmdOverwriteDec := TRUE ;
END_METHOD

METHOD PUBLIC CmdReset : BOOL
VAR_INPUT
END_VAR
// Set reset axis to true 				
	bExec_Reset 	:= TRUE ; 
	bInternalEnable	:= TRUE ;
	
// Check error state of axis
	bError 		:= AxisRef.Status.Error ; 

// Reset CmdMoveAbs
bResetCmdMoveAbs := TRUE;

// Set feedback output 
	CmdReset := (NOT bError);
END_METHOD

METHOD PUBLIC CmdSafeSpeed : BOOL
VAR_INPUT
END_VAR
// Set safestop command
bCmdSafeSpeed := TRUE ; 

// Set feedback output 
CmdSafeSpeed := fbMcPower.Override = fSafeOverride  ;
END_METHOD

METHOD PUBLIC CmdSafeStop : BOOL
VAR_INPUT
END_VAR
IF AxisRef.Status.Coupled THEN 
	CmdSafeStop := AxisRef.Status.NotMoving ;
	RETURN;
END_IF

// Set safestop command
bCmdSafeStop := TRUE ; 

// Set feedback output 
CmdSafeStop := bIsSafe OR NOT bInitOk;
END_METHOD

METHOD PUBLIC CmdSetPosition : BOOL
VAR_INPUT
	fPosition		: LREAL ; // encoder position
	bSetRelative	: BOOL 	; // TRUE = relative position offset, FALSE = Absolute position
END_VAR
// check if error is active
	IF bError THEN
		stFault.Active 			:= TRUE 						;
		stFault.Description		:= 'Call to CmdSetPosition while axis has an error';
		stFault.FaultType		:= E_FaultTypes.CF				;	
		RETURN;
	END_IF

bExec_SetPosition 			:= NOT fbMcSetPosition.Busy AND NOT fbMcSetPosition.Done ; 
fbMcSetPosition.Position	:= fPosition ;
fbMcSetPosition.Mode		:= bSetRelative ;

// Reset CmdMoveAbs
bResetCmdMoveAbs := TRUE;

CmdSetPosition := fbMcSetPosition.Done;
END_METHOD

METHOD PRIVATE ExecEnable : BOOL
VAR_INPUT
END_VAR
// ===== Set axis enable ======
IF NOT bSTOOK 
OR AxisRef.Status.DriveDeviceError
OR bExec_Reset THEN 
	bCmdEnableAxis 	:= FALSE ;
	bCmdManual 		:= FALSE ;
ELSIF bCmdManual THEN 
	bCmdEnableAxis 	:= TRUE ;
	bInternalEnable S= bCmdManual ;
	bCmdManual 		:= FALSE ;
ELSE 
	bCmdEnableAxis	:= bEnable ;
END_IF

// ===== Check if axis is bussy with a command =====
	bInternalEnable S= AxisRef.Status.HasJob;
	bInternalEnable	S= bIcfAlwaysEnable ; // always enable axis if configured
	bInternalEnable	S= AxisRef.Status.Coupled ;

// ===== Axis disable timer after last command =====
	TofIntAxisEnable (	IN:= bInternalEnable, PT := tDisableDelay);

// ===== Enable drive =====
	fbMcPower(	Axis			:= AxisRef , 
				Enable			:= bCmdEnableAxis AND TofIntAxisEnable.Q, 
				Enable_Positive	:= bIcfEnableForward, 
				Enable_Negative	:= bIcfEnableReverse, 
				BufferMode		:= MC_Buffered );  
				
// ===== Reset internal enable signal =====
	bInternalEnable := FALSE ; 	

// ===== Delayed enable function =====	
	IF fbMcPower.Enable AND fbMcPower.Status THEN
		bAxisIsEnabled := TRUE ;
	ELSIF NOT fbMcPower.Enable OR AxisRef.Status.Error THEN 
		bAxisIsEnabled := FALSE ; 
	END_IF

	TonMotionEnable	(IN := bAxisIsEnabled, PT := tEnableDelay);
	bDelayedEnable 	:= TonMotionEnable.Q ;	

IF AxisRef.Status.DriveDeviceError 
AND bCmdEnableAxis OR bCmdManual THEN
	bError					:= TRUE							;
	stFault.Active 			:= TRUE 						;
	stFault.Description		:= CONCAT('Drive device error ', UDINT_TO_STRING(AxisRef.Status.ErrorID));
	stFault.FaultType		:= E_FaultTypes.FF				;
ELSIF fbMcPower.Error THEN 
	bError					:= TRUE							;
	stFault.Active 			:= TRUE 						;
	stFault.Description		:= CONCAT('Enable Fault ', UDINT_TO_STRING(fbMcPower.ErrorID));
	stFault.FaultType		:= E_FaultTypes.FF				;
END_IF
END_METHOD

METHOD INTERNAL ExecGearDynamic : BOOL
VAR_INPUT
END_VAR
// ===== invert gear ratio if reverse slave is active =====
	IF bReverseSlave THEN 
		fbMcGearInDyn.GearRatio := fCmdGearRatio * -1 ;
	ELSE 
		fbMcGearInDyn.GearRatio := fCmdGearRatio ;
	END_IF

// ===== Execute gear in function =====
	fbMcGearInDyn ( 	Master 			:= refMasterAxis,
						Slave			:= AxisRef,
						Enable 			:= bExec_GearSlaveDyn AND bDelayedEnable,
						Acceleration	:= 0,
						Deceleration	:= 0	); 
						
// ===== reset command =====
	bExec_GearSlaveDyn	:= FALSE ;
	bGearedAsSlave		:= fbMcGearInDyn.InGear ; 

// Gearing fault handling 
	IF fbMcGearInDyn.Error THEN 
		bError					:= TRUE							;
		stFault.Active 			:= TRUE 						;
		stFault.Description		:= CONCAT('Gear dynamic Fault ', UDINT_TO_STRING(fbMcGearInDyn.ErrorID));	
		stFault.FaultType		:= E_FaultTypes.FF				;
	END_IF
END_METHOD

METHOD INTERNAL ExecGearIn : BOOL
VAR_INPUT
END_VAR
// ===== invert gear ratio if reverse slave is active =====
	IF bReverseSlave THEN 
		fbMcGearInSlave.RatioNumerator := fCmdGearRatio * -1 ;
	ELSE 
		fbMcGearInSlave.RatioNumerator := fCmdGearRatio ;
	END_IF

// ===== Execute gear in function =====
	fbMcGearInSlave ( 	Master 			:= refMasterAxis,
						Slave			:= AxisRef,
						Execute 		:= bExec_GearAsSlave AND bDelayedEnable,
						RatioDenominator:= 1,
						Acceleration	:= 0,
						Deceleration	:= 0	); 
						
// ===== reset command =====
	bExec_GearAsSlave 	:= FALSE  ;
	bGearedAsSlave		S= fbMcGearInSlave.InGear ; 

// Gearing fault handling 
	IF fbMcGearInSlave.Error THEN 
		bError					:= TRUE							;
		stFault.Active 			:= TRUE 						;
		stFault.Description		:= CONCAT('Gear as slave Fault ', UDINT_TO_STRING(fbMcGearInSlave.ErrorID));
		stFault.FaultType		:= E_FaultTypes.FF				;
	END_IF
END_METHOD

METHOD INTERNAL ExecGearOut : BOOL
VAR_INPUT
END_VAR
// ===== execute gear out function ======
	fbMcGearOutSlave (	Slave 	:= AxisRef,
						Execute := bExec_GearOutSlave );

// ===== reset command =====
	bExec_GearOutSlave	:= false ;
	bGearedAsSlave		R= fbMcGearOutSlave.Done 	; 

// Gearing fault handling 
	IF fbMcGearOutSlave.Error THEN 
		bError					:= TRUE							;
		stFault.Active 			:= TRUE 						;
		stFault.Description		:= CONCAT('Gear out Fault ', UDINT_TO_STRING(fbMcGearOutSlave.ErrorID));
		stFault.FaultType		:= E_FaultTypes.FF				;
	END_IF
END_METHOD

METHOD INTERNAL ExecHalt : BOOL
VAR_INPUT
END_VAR
// ==== Execute halt function ===== 
fbMcHalt (	Axis 		:= AxisRef,
			Execute 	:= bExec_Halt );

// ===== reset command =====
	bExec_Halt := FALSE ;
	
// Halt fault handling 
	IF fbMcHalt.Error THEN 
		bError					:= TRUE							;
		stFault.Active 			:= TRUE 						;
		stFault.Description		:= CONCAT('Halt Fault ', UDINT_TO_STRING(fbMcHalt.ErrorID));
		stFault.FaultType		:= E_FaultTypes.FF				;
	END_IF
END_METHOD

METHOD INTERNAL ExecHome : BOOL
VAR_INPUT
END_VAR
// ==== execute homing function =====
	IF bIcfNCHomeSensor THEN 
		fbmchome.bCalibrationCam	:= NOT IAxisHome;
	ELSE
		fbmchome.bCalibrationCam	:= IAxisHome;
	END_IF		
		
	fbMcHome(	Axis			:= AxisRef,
				Execute			:= bExec_Home AND bDelayedEnable,
				HomingMode		:= mcHomingMode ); 
			
// Reset exec command 
	bExec_Home 	:= FALSE ;
	bHomed		S= fbMcHome.Done;
				
// fault handling
// In manual mode, releasing the "Home" button before homing is finished
// will immediately trigger a 19210 homing error, setting the system to Fault state.
// Therefore, when in manual mode, the level of the error will be reduced to a warning.
	IF fbMcHome.Error THEN
		bResetCalibrationFlag	:= TRUE;
		bError					:= TRUE							;
		stFault.Active 			:= TRUE 						;
		stFault.Description		:= CONCAT('Homing Fault ', UDINT_TO_STRING(fbMcHome.ErrorID));
		IF bManual THEN
			stFault.FaultType		:= E_FaultTypes.OW				;
		ELSE
			stFault.FaultType		:= E_FaultTypes.FF				;
		END_IF
	END_IF
END_METHOD

METHOD INTERNAL ExecJog : BOOL
VAR_INPUT
END_VAR
// ===== Execute Jog function =====
	IF bCmdLimitVelocity THEN 
		fbMcJog.Velocity := MIN(fCmdVelocityLimit, fbMcJog.Velocity); 
	END_IF

	// function call
	fbMcJog (	Axis 		:= AxisRef,
				JogForward	:= bExec_JogPositive AND bDelayedEnable,
				JogBackwards:= bExec_JogNegative AND bDelayedEnable,
				Acceleration:= fAcceleration,
				Deceleration:= fDeceleration );

// ===== reset command =====
	bExec_JogPositive 	:= FALSE  ;
	bExec_JogNegative	:= FALSE  ;
	
// Jog fault handling 
	IF fbMcJog.Error THEN 
		bError					:= TRUE							;
		stFault.Active 			:= TRUE 						;
		stFault.Description		:= CONCAT('Jog Fault ', UDINT_TO_STRING(fbMcJog.ErrorID));
		stFault.FaultType		:= E_FaultTypes.FF				;
	END_IF
END_METHOD

METHOD INTERNAL ExecMoveAbsolute : BOOL
VAR_INPUT
END_VAR
// ==== execute move absolute function =====
FOR i := 0 TO 1 DO 
	// Limit velocity
	IF bCmdLimitVelocity THEN 
		fbMcJog.Velocity := MIN(fCmdVelocityLimit, fbMcMoveAbsolute[i].Velocity); 
	END_IF
	// function call
	fbMcMoveAbsolute[i](	Axis 		:= AxisRef,
							Execute 	:= arExec_MoveAbs[i] AND bDelayedEnable,
							Acceleration:= fAcceleration,
							Deceleration:= fDeceleration );  

	// If function is done then reset command values
	IF fbMcMoveAbsolute[i].Done OR fbMcMoveAbsolute[i].CommandAborted THEN 
		fbMcMoveAbsolute[i].Velocity	:= 0 ;
		fbMcMoveAbsolute[i].Position	:= 0 ; 
	END_IF

	// reset Exec command 
	arExec_MoveAbs[i] R= bDelayedEnable ; 
	
	// fault handling 
	IF fbMcMoveAbsolute[i].Error THEN 
		bError					:= TRUE							;
		stFault.Active 			:= TRUE 						;
		stFault.Description		:= CONCAT('Move absolute fault ', UDINT_TO_STRING(fbMcMoveAbsolute[i].ErrorID));
		stFault.FaultType		:= E_FaultTypes.FF				;
	END_IF
END_FOR
END_METHOD

METHOD INTERNAL ExecMoveModulo : BOOL
VAR_INPUT
END_VAR


// ===== Execute move modulo function =====
FOR i := 0 TO 1 DO 
	IF bCmdLimitVelocity THEN 
		fbMcJog.Velocity := MIN(fCmdVelocityLimit, fbMcMoveModulo[i].Velocity); 
	END_IF
	// function call
	fbMcMoveModulo[i](	Axis 		:= AxisRef,
						Execute 	:= arExec_MoveModulo[i] AND bDelayedEnable,
						Acceleration:= fAcceleration,
						Deceleration:= fDeceleration);  
	
	// If function is done then reset command values
	IF fbMcMoveModulo[i].Done OR fbMcMoveModulo[i].CommandAborted OR NOT arExec_MoveModulo[i] THEN 
		fbMcMoveModulo[i].Velocity	:= 0 ;
		fbMcMoveModulo[i].Position	:= 0 ; 
	END_IF

	// reset Exec command 
	arExec_MoveModulo[i] := FALSE ; 
	
	// fault handling 
	IF fbMcMoveModulo[i].Error THEN 
		bError					:= TRUE							;
		stFault.Active 			:= TRUE 						;
		stFault.Description		:= CONCAT('Move module Fault ', UDINT_TO_STRING(fbMcMoveModulo[i].ErrorID));
		stFault.FaultType		:= E_FaultTypes.FF			;
	END_IF
END_FOR
END_METHOD

METHOD INTERNAL ExecMoveRelative : BOOL
VAR_INPUT
END_VAR
//ReCmd_MoveModulo(CLK := bCmd_MoveModulo );
//bCmd_MoveModulo	:= FALSE ;

// ===== Execute move relative function ======
FOR i := 0 TO 1 DO 
	// Limit velocity
	IF bCmdLimitVelocity THEN 
		fbMcJog.Velocity := MIN(fCmdVelocityLimit, fbMcMoveModulo[i].Velocity); 
	END_IF
	// function call
	fbMCMoveRelative[i](	Axis 		:= AxisRef,
							Execute		:= arExec_MoveRelative[i] AND bDelayedEnable,
							Acceleration:= fAcceleration,
							Deceleration:= fDeceleration );

	// If function is done then reset command values
	IF fbMCMoveRelative[i].Done OR fbMCMoveRelative[i].CommandAborted OR NOT arExec_MoveRelative[i] THEN 
		fbMCMoveRelative[i].Velocity	:= 0 ;
		fbMCMoveRelative[i].Distance	:= 0 ; 
	END_IF

	// reset Exec command 
	arExec_MoveRelative[i] := FALSE ; 
	
	// fault handling 
	IF fbMCMoveRelative[i].Error THEN 
		bError					:= TRUE							;
		stFault.Active 			:= TRUE 						;
		stFault.Description		:= CONCAT('Move relative Fault ', UDINT_TO_STRING(fbMCMoveRelative[i].ErrorID));
		stFault.FaultType		:= E_FaultTypes.FF			;
	END_IF
END_FOR
END_METHOD

METHOD INTERNAL ExecMoveVelocity : BOOL
VAR_INPUT
END_VAR
// ===== Execute move velocity function =====
	IF bCmdLimitVelocity THEN 
		fbMcJog.Velocity := MIN(fCmdVelocityLimit, fbMcMoveVelocity.Velocity); 
	END_IF

// function call
fbMcMoveVelocity (	Axis 		:= AxisRef,
					Execute		:= (bExec_MoveVelocity OR bExec_MoveVelocityDynamic) AND bDelayedEnable,
					Acceleration:= fAcceleration,
					Deceleration:= fDeceleration );

// ===== reset command =====
bExec_MoveVelocity 			:= FALSE ;
bExec_MoveVelocityDynamic 	:= FALSE;
	
// Halt fault handling 
IF fbMcMoveVelocity.Error THEN 
	bError					:= TRUE							;
	stFault.Active 			:= TRUE 						;
	stFault.Description		:= CONCAT('Move velocity Fault ', UDINT_TO_STRING(fbMcMoveVelocity.ErrorID));
	stFault.FaultType		:= E_FaultTypes.FF				;
END_IF
END_METHOD

METHOD INTERNAL ExecReadStatus : BOOL
VAR_INPUT
END_VAR
AxisRef.ReadStatus();
					
// convert velocity to RPM for output if aplicable
IF bIcfCmdVelocityRpm THEN 
	fVelocity := AxisRef.NcToPlc.ActVelo / 6 ;
ELSE 
	fVelocity := AxisRef.NcToPlc.ActVelo ;
END_IF

// write position output
IF bIcfModuloAxis THEN 
	fActPosition := AxisRef.NcToPlc.ModuloActPos ;
ELSE
	fActPosition := AxisRef.NcToPlc.ActPos ;
END_IF
						
// set status bits 
bIdle := NOT AxisRef.Status.HasJob ;

// In position 
	rtrigInPosition( 	CLK := AxisRef.Status.InTargetPosition, 
						Q => bReInTargetPos);
END_METHOD

METHOD INTERNAL ExecReset : BOOL
VAR_INPUT
END_VAR
VAR
	xMcReset			: BOOL ; // Execute MC reset
	xSoeReset			: BOOL ; // Execute SOE reset

END_VAR
//IF  AxisRef.Status.Moving AND bExec_Reset THEN // If the axis is still moving execute safe stop first
//	RETURN;
IF AxisRef.Status.Coupled THEN 
	bResetDone 	:= NOT AxisRef.Status.Error;
	bExec_Reset	R= bResetDone  ;
	RETURN;
END_IF

// ===== reset command =====
	bExec_Reset	R= fbMcReset.Done  ;

// ==== execute reset functions =====
IF AxisRef.Status.DriveDeviceError AND IAxisSTOOK THEN 
		xSoeReset := TRUE ;
ELSIF bSTOOK AND bExec_Reset THEN
		xMcReset	:= TRUE ;
ELSE 
	xSoeReset 	:= FALSE ;
	xMcReset	:= FALSE ;
END_IF

fbSoeReset	( 	Execute := xSoeReset,
				Timeout	:= T#5S,
				Axis	:= AxisRef);

fbMcReset	( 	Execute	:= xMcReset,
				Axis	:= AxisRef ); 
				
// ===== Set feedback =====
	bResetDone 	S= fbMcReset.Done  ;
	bResetDone	R= AxisRef.Status.Error ;
	tonResetDone (IN	:= bResetDone);

// ===== reset limitations =====
	bCmdSafeSpeed 	:= FALSE ;

	
// Reset fault handling 
	IF fbSoeReset.Error OR fbMcReset.Error THEN 
		bError					:= TRUE							;
		stFault.Active 			:= TRUE 						;
		stFault.Description		:= CONCAT('Reset Fault ', UDINT_TO_STRING(fbMcReset.ErrorID));
		stFault.FaultType		:= E_FaultTypes.FF				;
	END_IF
END_METHOD

METHOD PRIVATE ExecSafeFunctions : BOOL
VAR_INPUT
END_VAR
// ===== Safe torque off function =====
	IF bIcfSTOPresent THEN 
		tonSTOOK(IN := IAxisSTOOK, PT := T#1000MS);
		bSTOOK := tonSTOOK.Q AND NOT AxisRef.Status.DriveDeviceError;
//		bSTOOK	:= IAxisSTOOK ;
	ELSE 
		bSTOOK := true ;
	END_IF
	
// ==== Safe operation functions (overrule all other motion functions) =====
	IF NOT AxisRef.Status.Coupled AND bSTOOK THEN 
		fbMcStop( 	Axis 			:= AxisRef		,
					Execute 		:= bCmdSafeStop AND NOT bExec_Reset,
					Deceleration	:= fMaxDec		);
	END_IF
	
	// Reset axis command			
	bCmdSafeStop 	R= fbMcStop.Done OR AxisRef.Status.HasBeenStopped OR NOT bSTOOK ;
	bStopped		:= AxisRef.Status.HasBeenStopped OR NOT bSTOOK ;

// Safestop fault handling 
	IF fbMcStop.Error THEN 
		bError					:= TRUE							;
		stFault.Active 			:= TRUE 						;
		stFault.Description		:= CONCAT('Safe stop axis fault ', UDINT_TO_STRING(fbMcStop.ErrorID));
		stFault.FaultType		:= E_FaultTypes.FF				;
	END_IF
	
// ===== Safe speed monitoring =====
	IF bCmdSafeSpeed THEN 
		fbMcPower.Override 	:= fSafeOverride ;
		bCmdSafeSpeed		:= FALSE ;
	ELSE 
		fbMcPower.Override := 100 ;
	END_IF

// ===== Dev is safe feedback =====
bIsSafe := AxisRef.Status.HasBeenStopped OR AxisRef.Status.Disabled  ;
END_METHOD

METHOD INTERNAL ExecSetPosition : BOOL
VAR_INPUT
END_VAR
// ====== set position of axis ======
IF bExec_SetPosition OR fbMcSetPosition.Busy THEN 
	fbMcSetPosition (	Axis 	:= AxisRef,
						Execute	:= bExec_SetPosition );
	bExec_SetPosition := TRUE ;
END_IF
END_METHOD

METHOD PRIVATE ExecWriteParameter : BOOL
VAR_INPUT
END_VAR
// check if axis is disabled before writeing parameter
	AxisRef.ReadStatus();
	IF AxisRef.Status.Disabled 
	AND (fbMcWriteParameter.Busy OR bExec_ParWritePers) THEN
		fbMcWriteParameter	( 	Axis 	:= AxisRef,
								Execute	:= bExec_ParWritePers );
	ELSE
		fbMcWriteParameter.Execute := FALSE ; 
		RETURN;
	END_IF
						
// fault handling 
	IF fbMcWriteParameter.Error THEN 
		bError					:= TRUE							;
		stFault.Active 			:= TRUE 						;
		stFault.MessageNumber	:= E_MessageNumbers.FF_AxisFault;
		stFault.Description		:= CONCAT('Cannot write parameter Id#:', UDINT_TO_STRING(fbMcHome.ErrorID));
		stFault.Description		:= CONCAT( sName , stfault.Description ) ;
		stFault.FaultType		:= E_FaultTypes.FF				;
	END_IF
 
// reset commands
	bExec_ParWritePers := FALSE ;
END_METHOD

METHOD PUBLIC Init : BOOL
VAR_INPUT
	// Message location data
	nId			: UINT ; // Identification number of object
	nParentId	: UDINT ; // Id of higher level If aplicable (0 = no parent)
	// Config Bits
	bIcfCmdVelocityRpm	: BOOL := FALSE ; // input speeds in Rpm
	bIcfEnableForward 	: BOOL := TRUE 	; // Enable forward motion
	bIcfEnableReverse	: BOOL := TRUE 	; // Enable reverse motion
	bIcfAlwaysEnable	: BOOL := FALSE ; // 1 = Axis always enabled, 0 = Axis disabled at Idle 
	bIcfModuloAxis		: BOOL := FALSE ; // Show axis position as modulo
	bIcfSTOPresent		: BOOL := FALSE ; // Axis safe torque off is present
	bIcfNCHomeSensor	: BOOL := FALSE ; // Homing sensor is inverted (NC)	
	// Config Values 
	mcHomingMode 		: MC_HomingMode := MC_HomingMode.MC_DefaultHoming; 
	fSafeOverride		: LREAL := 10	; // Safe velocity override [%]
	nEncTurnoverVal 	: LREAL := 360	; // encoder turnover value 
	tEnableDelay		: time 	:= T#0MS; // Time between axis enable command and motion command execution (0 := no delay active)	
	tDisabledelay		: TIME 	:= T#100MS; // Axis idle time before axis is disabled 
END_VAR
VAR 
	bActVeloReadValid 	: BOOL ; // velocity parameter read is valid 
	bActAccReadValid 	: BOOL ; // Acceleration parameter read is valid 
	bActDecReadValid 	: BOOL ; // Deceleration parameter read is valid 
	bActParamValid 		: BOOL ; // Parameter read is valid 
END_VAR
// ====== Set init to true =====
	bInitOk	:= TRUE ; 

// ====== Calculate device id =====
	bInitOk :=	ExecIdentifyDevice(nId,nParentId, E_ComponentTypes.Axis) AND bInitOk;

// ====== Set manual device type ======
	eDevType := E_Devices.Axis ;	
	
// ===== Read system configuration =====
	McReadSysVelo	(	Axis 			:= AxisRef,
						Enable 			:= Cmd_EnDriveParRead ,
						ParameterNumber := MaxVelocitySystem ,
						ReadMode		:= 1,
						Valid			=> bActVeloReadValid ,						
						Busy			=> ,
						Error			=> ,
						ErrorID			=> ,
						Value			=> fMaxVelo );
	McReadSysAcc	(	Axis 			:= AxisRef,
						Enable 			:= Cmd_EnDriveParRead ,
						ParameterNumber := MaxAccelerationSystem ,
						ReadMode		:= 1,
						Valid			=> bActAccReadValid ,						
						Busy			=> ,
						Error			=> ,
						ErrorID			=> ,
						Value			=> fMaxAcc );
	McReadSysDec	(	Axis 			:= AxisRef,
						Enable 			:= Cmd_EnDriveParRead ,
						ParameterNumber := MaxDecelerationSystem ,
						ReadMode		:= 1,
						Valid			=> bActDecReadValid ,						
						Busy			=> ,
						Error			=> ,
						ErrorID			=> ,
						Value			=> fMaxDec );

	IF 	fMaxVelo > 0 
	AND fMaxAcc >0
	AND fMaxDec >0 THEN 
		bActParamValid	:= TRUE ; 
		fCmdAcc 		:= fMaxAcc * 0.9;
		fCmdDec		:= fMaxDec * 0.9;
	END_IF

	IF NOT Cmd_EnDriveParRead AND NOT bActParamValid THEN  
		Cmd_EnDriveParRead := TRUE;
	ELSIF Cmd_EnDriveParRead THEN
		Cmd_EnDriveParRead := FALSE;
	END_IF

// ===== Configure Axis =====
	// ***** Config Bits *****
		THIS^.bIcfCmdVelocityRpm	:= bIcfCmdVelocityRpm	; // Enable speed inputs in Rpm
		THIS^.bIcfEnableForward 	:= bIcfEnableForward 	; // Enable forward motion
		THIS^.bIcfEnableReverse		:= bIcfEnableReverse	; // Enable reverse motion
		THIS^.bIcfAlwaysEnable		:= bIcfAlwaysEnable		; // Always enable motor and brake if safety is ok
		THIS^.bIcfModuloAxis		:= bIcfModuloAxis		; // show axis position as modulo
		THIS^.bIcfSTOPresent		:= bIcfSTOPresent		; // Axis has safe torque off function
		THIS^.bIcfNCHomeSensor		:= bIcfNCHomeSensor		; // Axis homing sensor is NC	
	// ***** config homing Mode ***** 
 		THIS^.mcHomingMode 			:= mcHomingMode ; // set homing mode
	// ***** Velocity settings *****
		THIS^.fSafeOverride			:= fSafeOverride	; 	
	// ***** Encoder values *****
		THIS^.fEncoderTurnoverValue := nEncTurnoverVal	; // turnover value for encoder = 25.6 mm per rev * 4096 revolutions 
	// ***** Time delay enable off *****
		THIS^.tEnableDelay		:= tEnableDelay	;
		THIS^.tDisableDelay 	:= tDisabledelay ;		
		
// ===== configure parameters =====
	ParHomeOffset.fMinimum 		:= -1E7;
	ParHomeOffset.fMaximum		:= 1E7;
	ParHomeOffset.nNumber 		:= stIdentity.nLocationId + 1;
	ParHomeOffset.sDiscription  := CONCAT( STR1 := stIdentity.sName, STR2 := ' home position offset');
	ParHomeOffset.sName			:= CONCAT( STR1 := stIdentity.sName, STR2 := ' Home position offset');
	ParHomeOffset.sType			:= 'MPar';
	ParHomeOffset.sUnit			:= 'unit';
	refFbParHandler.CmdAddParameter( refParameter := ParHomeOffset );

// ===== reset axis state indicators ======
	bError 	:= FALSE;

// ====== Set init to done =======
bInitOk := bActParamValid AND bInitOk;
Init := bInitOk;
END_METHOD

END_FUNCTION_BLOCK

// ---- BaseFunctions/FB_DevBase.TcPOU
{attribute 'reflection'}
FUNCTION_BLOCK PUBLIC FB_DevBase EXTENDS FB_FunctionBase
VAR_INPUT
	bEmbedded		: BOOL 	:= FALSE ; // Device is embedded into another device (not added to manual screen)
	// function references 
	refFbManualCtrl	: REFERENCE TO FB_ManualController := GVL_Devices.fbManualController; // reference to manual handler
END_VAR
VAR_OUTPUT
	eDevType		: E_Devices		:= E_Devices.Undefined	; // Type of Device 	
END_VAR
VAR
	// Manual control variables
	bAddedToManual	: BOOL 	:= FALSE 	; // device is added tot manual control function 	
END_VAR

SUPER^();

// Add device to manual screen
IF NOT bEmbedded THEN 
	IF bInitOk
	AND NOT bAddedToManual 
	AND __ISVALIDREF(refFbManualCtrl)
	THEN 
		bAddedToManual S= refFbManualCtrl.CmdAddDevice(THIS^);
	END_IF
END_IF

METHOD PUBLIC CmdSafeStop : BOOL
VAR_INPUT
END_VAR
// check if device is safe
bIsSafe 	:= TRUE;
CmdSafeStop := bIsSafe ;
END_METHOD

END_FUNCTION_BLOCK

// ---- GroupHandlers/ManualControlHandler/FB_ManualController.TcPOU
FUNCTION_BLOCK FB_ManualController
VAR_INPUT
	bBlockManualMode : BOOL; // Block (do not allow) manual mode 
END_VAR
VAR_OUTPUT
	bActive : BOOL; // TRUE if manual control is active
END_VAR
VAR
	stHMI				: UDT_HMI_ManualControl; // Link between FB and HMI
	
	nNumberOfDevices	: UDINT := 0; // Number of devices in DeviceArray
	nSelectedDevicePrev : UDINT := 0; // Previously selected device in HMI (array index)
 
	fbNodevice			: FB_DevBase; // Dummy to make all pointers point to a valid device
	stNoDevice			: UDT_DeviceID := (sName := 'No device', sType := TO_STRING(E_Devices.Undefined), pFunction := ADR(fbNodevice)); 

	arDeviceArray		: ARRAY [0..100] OF UDT_DeviceID := [stNoDevice];
END_VAR

stHMI.bBlocked := bBlockManualMode;
IF bBlockManualMode THEN
	stHMI.bEnabled := FALSE;
	stHMI.bReset := FALSE;
END_IF

bActive := stHMI.bEnabled;
IF bActive THEN
	// NOTE: The device is responsibe for disabling the manual mode when CmdManual is no longer called
	stHMI.refSelectedDevice.CmdManual();
END_IF

IF stHMI.nSelectedDevice <> nSelectedDevicePrev THEN // User changed device selection in the HMI
	// Get a reference to the selected device	
	stHMI.refSelectedDevice REF= arDeviceArray[stHMI.nSelectedDevice].pFunction^;
	
	// Remember previous selection
	nSelectedDevicePrev := stHMI.nSelectedDevice;

	// Update HMI frame (contains device specific manual controls)  
	CASE stHMI.refSelectedDevice.eDevType OF
		E_Devices.Valve:
			stHMI.pDevValve 			:= ADR(stHMI.refSelectedDevice);
		E_Devices.Cylinder:
			stHMI.pDevCylinder			:= ADR(stHMI.refSelectedDevice);
		E_Devices.Axis:
			stHMI.pDevAxis				:= ADR(stHMI.refSelectedDevice);
		E_Devices.PushButtonLight:
			stHMI.pDevPBL				:= ADR(stHMI.refSelectedDevice);
		E_Devices.DigitalSensor:
			stHMI.pDevDigitalInput		:= ADR(stHMI.refSelectedDevice);
		E_Devices.AnalogSensor:
			stHMI.pDevAnalogInput 		:= ADR(stHMI.refSelectedDevice);
		E_Devices.DigitalOut:
			stHMI.pDevDigitalOut		:= ADR(stHMI.refSelectedDevice);
		E_Devices.AnalogOut:
			stHMI.pDevAnalogOut			:= ADR(stHMI.refSelectedDevice);
		E_Devices.PWMController:
			stHMI.pDevPWMController		:= ADR(stHMI.refSelectedDevice);
		E_Devices.DoublePWMController:
			stHMI.pDevDoublePWM			:= ADR(stHMI.refSelectedDevice);
		E_Devices.Encoder:
			stHMI.pDevEncoder			:= ADR(stHMI.refSelectedDevice);
		E_Devices.AnalogAxis:
			stHMI.pDevAnalogAxis		:= ADR(stHMI.refSelectedDevice);
		E_Devices.TwoVelocityAxis:
			stHMI.pDevTwoVelocityAxis 	:= ADR(stHMI.refSelectedDevice);
		E_Devices.KL5151:
			stHMI.pDevKL5151			:= ADR(stHMI.refSelectedDevice);
		E_Devices.KL1512:
			stHMI.pDevKL1512			:= ADR(stHMI.refSelectedDevice);
	END_CASE

END_IF

// Reset device 
IF stHMI.bReset THEN
	stHMI.bReset R= stHMI.refSelectedDevice.CmdReset();
END_IF

METHOD PUBLIC CmdAddDevice : BOOL
VAR_INPUT
	refToDevice	: REFERENCE TO FB_DevBase ;
END_VAR
VAR
	bDevAdded : BOOL ;
	i : UDINT; // Iterator
	nArraySize : UINT;
END_VAR
// Check if device is not already in the array 
FOR i:= 0 TO nNumberOfDevices DO 
	IF arDeviceArray[i].sName = refToDevice.stIdentity.sName THEN 
		bDevAdded := TRUE ;
	END_IF 
END_FOR

// If device is not found add device to the list
IF NOT bDevAdded THEN 
	nArraySize := SIZEOF(arDeviceArray) / SIZEOF(arDeviceArray[0]);
	nNumberOfDevices := LIMIT(0, nNumberOfDevices + 1, nArraySize);
	arDeviceArray[nNumberOfDevices].sType 		:= TO_STRING(refToDevice.eDevType)	;
	arDeviceArray[nNumberOfDevices].sName		:= refToDevice.stIdentity.sName	;
	arDeviceArray[nNumberOfDevices].pFunction 	:= ADR(refToDevice)		;	
	bDevAdded := TRUE ;
END_IF

CmdAddDevice := bDevAdded ;
END_METHOD

METHOD FB_init : BOOL
VAR_INPUT
	bInitRetains : BOOL; // if TRUE, the retain variables are initialized (warm start / cold start)
	bInCopyCode : BOOL;  // if TRUE, the instance afterwards gets moved into the copy code (online change)
END_VAR
// Assure stHMI always has valid references
stHMI.refSelectedDevice REF= THIS^.fbNodevice;
END_METHOD

END_FUNCTION_BLOCK

// ---- _TESTS/PRG_TEST_FB_DEVVALVE.TcPOU
PROGRAM INTERNAL PRG_TEST_FB_DEVVALVE
VAR
	bEnableTests : BOOL;
	
	fbDevValve : Fb_DevValve;
	
	// Settings
	eResetState : E_ValveResetState;
	eSafeState : E_ValveResetState;
	
	// Public commands
	bInit : BOOL;
	bCmdClose : BOOL;
	bCmdHold : BOOL;
	bCmdManual : BOOL;
	bCmdOpen : BOOL;
	bCmdReset : BOOL;
	bCmdSafeStop : BOOL;
	bCmdSafeStop_RetVal : BOOL;
	bCmdTeach : BOOL;
	
//	// Inputs
//	bFco_Closed	: BOOL;
//	bFco_Open	: BOOL;
	
//	// Outputs
//	q_Open : BOOL;
//	q_Close : BOOL;
END_VAR

IF bEnableTests THEN
	fbDevValve();

	IF bInit THEN
		bInit R= fbDevValve.Init(
			nId			:= 1, 
			nParentId	:= 0,
			eResetState	:= eResetState,
			eSafeState	:= eSafeState
		);
	END_IF

	IF bCmdClose THEN bCmdClose R= fbDevValve.CmdClose(); END_IF
	IF bCmdHold THEN fbDevValve.CmdHold(); END_IF
	IF bCmdManual THEN fbDevValve.CmdManual(); END_IF
	IF bCmdOpen THEN bCmdOpen R= fbDevValve.CmdOpen(); END_IF
	IF bCmdReset THEN bCmdReset R= fbDevValve.CmdReset(); END_IF
	IF bCmdSafeStop THEN bCmdSafeStop_RetVal := fbDevValve.CmdSafeStop(); END_IF
	IF bCmdTeach THEN fbDevValve.CmdTeach(); END_IF
END_IF

END_PROGRAM

// ---- Actuators/Cylinder/Functions/FB_DevValve.TcPOU
{attribute 'reflection'}
FUNCTION_BLOCK PUBLIC FB_DevValve EXTENDS FB_DevBase
VAR_INPUT
	// Manual control 
	stManualCtrl	: UDT_ManualValveControl ;
END_VAR
VAR_OUTPUT
	// ===== Status indicators =======
	bFco_Closed		:	BOOL := FALSE ;
	bFco_Open		: 	BOOL := FALSE ;
	fTimeToOpen		: 	LREAL ;
	fTimeToClose	: 	LREAL ;
END_VAR
VAR
	// Pararmeters
		stParTimeToClose	: Udt_Parameter := (fValue := 50) ; // time to close parameter
		stParTimeToOpen		: Udt_Parameter	:= (fValue := 50) ; // Time to open parameter
	// Hardware links 
		q_Open			AT %Q* : BOOL := FALSE 	; // Open valve
		q_Close 		AT %Q* : BOOL := FALSE	; // Close valve
	// Internal commands
		bCmdClose 	: BOOL := FALSE ; // close valve 
		bCmdOpen	: BOOL := FALSE ; // Open valve
		bCmdHold	: BOOL := FALSE ; // Hold valve status change
		bCmdSafeStopCallActive : BOOL; // Method CmdSafeStop is being called 
	// Time functions 
		fbTOnClose	: TON	; // Timer for valve close
		FbTOnOpen	: TON 	; // Timer for valve Open
		fbTimerSwitchDir: TON ; // Time for teach function switch direction 
	// reset and safe state
		eResetState		: E_ValveResetState := 0		; // Cylinder reset state variable (default is idle) 
		eSafeState		: E_ValveResetState	:= 0		; // Valve safe state
END_VAR

// set device type
IF eDevType = E_Devices.Undefined THEN 
	eDevType := E_Devices.Valve ;
END_IF

// Call base function
	SUPER^();

// ===== hold all actions if not initialized ======
IF NOT bInitOk THEN
	RETURN;
END_IF 

// ====== Set Outputs =======
	ExecSetOutPuts();

// ===== collect feedback ======
	ExecSetFeedback();

METHOD PUBLIC CmdClose : BOOL // close valve or retract cylinder
VAR_INPUT
END_VAR
IF bManual THEN 
	RETURN;
END_IF

// ====== Set close command if enabled ======
	bCmdClose 	:= TRUE	;		
	bCmdOpen 	:= FALSE;

// ====== Check if command is blocked =====
	bBlockedCommand := bCmdHold;
	
// ===== Set feedback ======
	CmdClose := bFco_Closed ;
END_METHOD

METHOD PUBLIC CmdHold : BOOL
VAR_INPUT
END_VAR
// ====== set hold command =====
	bCmdHold := TRUE ;

CmdHold := bBlockedCommand ;
END_METHOD

METHOD PUBLIC CmdManual : BOOL
VAR_IN_OUT
END_VAR
// Enable manual commands
SUPER^.CmdManual();

// execute manual command 
	IF stManualCtrl.bCmdOpen THEN 
		bCmdClose 	:= FALSE;		
		bCmdOpen 	:= TRUE	;
	ELSIF stManualCtrl.bCmdClose THEN 
		bCmdClose 	:= TRUE	;		
		bCmdOpen 	:= FALSE;
	ELSIF stManualCtrl.bCmdTeach THEN
		CmdTeach ();
	END_IF
END_METHOD

METHOD PUBLIC CmdOpen : BOOL // Open valve or retract cylinder
VAR_INPUT
END_VAR
IF bManual THEN 
	RETURN;
END_IF

// ====== Set open command if enabled ======
	bCmdClose 	:= FALSE;		
	bCmdOpen 	:= TRUE	;

// ====== Check if command is blocked =====
	bBlockedCommand := bCmdHold;
	
// ===== Set feedback ======
	CmdOpen := bFco_Open ;
END_METHOD

METHOD PUBLIC CmdReset : BOOL
VAR_INPUT
END_VAR
// ====== Set outputs according to reset state =======
	IF bEnable THEN 
		CASE eResetState OF 
			E_ValveResetState.Res_Idle:
				bCmdClose 	:= FALSE;		
				bCmdOpen 	:= FALSE;
			E_ValveResetState.Res_Closed:
				bCmdClose 	:= TRUE	;		
				bCmdOpen 	:= FALSE;
			E_ValveResetState.Res_Open:
				bCmdClose 	:= FALSE;		
				bCmdOpen 	:= TRUE	;
		ELSE
			;
		END_CASE
	END_IF
// ======= Reset Error bit ======
	bErrorActive 	:= FALSE;
	bBusy			:= FALSE;
	
// ======= set feedback =======
	CmdReset := TRUE ;
END_METHOD

METHOD PUBLIC CmdSafeStop : BOOL
VAR_INPUT
END_VAR
bCmdSafeStopCallActive := TRUE;
bCmdOpen := FALSE ;
bCmdClose:= FALSE ;

CASE eSafeState OF 
	E_ValveResetState.Res_Idle:
		q_Close	:= bFco_Closed;		
		q_Open 	:= bFco_Open;
		bIsSafe := TRUE ;
	E_ValveResetState.Res_Closed:
		q_Close := TRUE ;
		q_Open  := FALSE ;
		bIsSafe := bFco_Closed OR NOT bFco_Open ;
	E_ValveResetState.Res_Open:
		q_Close := FALSE ;
		q_Open  := TRUE ;
		bIsSafe := bFco_Open OR NOT bFco_Closed;
END_CASE

CmdSafeStop := bIsSafe OR NOT bInitOk ;
END_METHOD

METHOD PUBLIC CmdTeach : BOOL
VAR_INPUT
END_VAR
// ====== teach cylinder from hardware inputs ======
	fbTimerSwitchDir(PT:= T#1S); 
// ===== Start test loop =====
IF bFco_Closed AND fbTimerSwitchDir.Q THEN
	bCmdClose 			:= FALSE;
	bCmdOpen 			:= TRUE ;
	fbTimerSwitchDir.IN	:= FALSE; 
ELSIF bFco_Open AND fbTimerSwitchDir.Q THEN
	bCmdClose 			:= TRUE ;
	bCmdOpen 			:= FALSE;
	fbTimerSwitchDir.IN	:= FALSE; 
ELSIF NOT bCmdClose AND NOT bCmdOpen THEN 
	bCmdClose 			:= TRUE ;
	bCmdOpen 			:= FALSE;
END_IF

// ====== start timing ========
	IF bCmdClose AND bFco_Closed THEN 
		fbTimerSwitchDir.IN := TRUE 		;
	ELSIF bCmdOpen AND bFco_Open THEN 
		fbTimerSwitchDir.IN := TRUE 		;
	END_IF
END_METHOD

METHOD PROTECTED ExecSetFeedback : BOOL
VAR_INPUT
END_VAR
// ====== Set timers =======
	fbTOnClose	(PT 	:= LREAL_TO_TIME(stParTimeToClose.fValue))	;
	FbTOnOpen	(PT		:= LREAL_TO_TIME(stParTimeToOpen.fValue))	;

// ====== Set timed feedback ======
	IF q_Close THEN 
		fbTOnClose.IN 	:= TRUE ;
		fbTOnopen.IN 	:= FALSE;
	ELSIF q_Open THEN 
		fbTOnClose.IN 	:= FALSE;
		FbTOnOpen.IN	:= TRUE ;
	ELSE 
		fbTOnClose.IN 	:= FALSE;
		FbTOnOpen.IN	:= FALSE;
	END_IF
	
// ====== set outputs =======
	bFco_Closed := fbTOnClose.Q ;
	bFco_Open	:= FbTOnOpen.Q	;
	bReady		:= bFco_Closed OR bFco_Open ;
	
// ====== Timer values =====
	fTimeToClose	:= stParTimeToClose.fValue;
	fTimeToOpen		:= stParTimeToOpen.fValue;
END_METHOD

METHOD PROTECTED ExecSetOutPuts : BOOL
VAR_INPUT
END_VAR
// ======= Set Outputs according to commands =======
IF NOT bCmdSafeStopCallActive
	AND NOT bCmdHold 
	AND (bEnable OR bManual) 	
THEN  
	q_Close	:= bCmdClose;
	q_Open	:= bCmdOpen	;
END_IF

// Reset manual and hold commands
bCmdHold 	:= FALSE ;
bCmdManual 	:= FALSE ;

bCmdSafeStopCallActive := FALSE; // Will be set to TRUE if CmdSafeStop is called
END_METHOD

METHOD PUBLIC Init : BOOL
VAR_INPUT
	// Messagedata 
	nId			: UINT ; // Identification number of object
	nParentId	: UDINT ; // Id of higher level If aplicable (0 = no parent)

	// Command state
	eResetState		: E_ValveResetState := 0		; // Cylinder reset state variable (default is idle) 
	eSafeState		: E_ValveResetState	:= 0		; // Valve safe state
END_VAR
// ====== Set init to true =====
	bInitOk	:= TRUE ; 

// ====== Calculate device id =====
	bInitOk :=	ExecIdentifyDevice(nId, nParentId, E_ComponentTypes.Cylinder) AND bInitOk;
	
// ====== Set outputs according to reset state =======
	THIS^.eResetState 	:= eResetState 	;
	THIS^.eSafeState	:= eSafeState	;	

	IF bEnable THEN 
		CASE eResetState OF 
			E_ValveResetState.Res_Idle:
				bCmdClose 	:= bFco_Closed	;		
				bCmdOpen 	:= bFco_Open	;
			E_ValveResetState.Res_Closed:
				bCmdClose 	:= TRUE;		
				bCmdOpen 	:= FALSE;
			E_ValveResetState.Res_Open:
				bCmdClose 	:= FALSE;		
				bCmdOpen 	:= TRUE ;
		END_CASE
	END_IF
// ======= Reset Error bit ======
	bErrorActive 	:= FALSE;
	bBusy			:= FALSE;

// ===== Set device type for manual control =====
	eDevType := E_Devices.Valve ;
	
// ===== configure parameters =====
	stParTimeToClose.fMinimum 		:= 0 		;
	stParTimeToClose.fMaximum		:= 60000 	;
	stParTimeToClose.nNumber 		:= stIdentity.nLocationId + 1;
	stParTimeToClose.sDiscription  	:= CONCAT( STR1 := stIdentity.sName, STR2 := ' average time it takes for the valve to close');
	stParTimeToClose.sName			:= CONCAT( STR1 := stIdentity.sName, STR2 := ' time to close');
	stParTimeToClose.sType			:= 'CPar';
	stParTimeToClose.sUnit			:= 'ms';

	stParTimeToOpen.fMinimum 		:= 0 		;
	stParTimeToOpen.fMaximum		:= 60000 	;
	stParTimeToOpen.nNumber 		:= stIdentity.nLocationId + 2;
	stParTimeToOpen.sDiscription  	:= CONCAT( STR1 := stIdentity.sName, STR2 := ' average time it takes for the valve to open');
	stParTimeToOpen.sName			:= CONCAT( STR1 := stIdentity.sName, STR2 := ' time to open');
	stParTimeToOpen.sType			:= 'CPar';
	stParTimeToOpen.sUnit			:= 'ms';
	
	// add parameters to handler 
	refFbParHandler.CmdAddParameter( refParameter := stParTimeToClose );
	refFbParHandler.CmdAddParameter( refParameter := stParTimeToOpen );

// Set feedback
Init := bInitOk;
END_METHOD

END_FUNCTION_BLOCK

// ---- _TESTS/PRG_TEST_FB_MANUALCONTROLLER.TcPOU
PROGRAM INTERNAL PRG_TEST_FB_MANUALCONTROLLER
VAR
	bEnableTests : BOOL;

	bInitDone 			: BOOL;
	fbManualController 	: FB_ManualController;
	fbDevValve 			: FB_DevValve;
END_VAR

IF bEnableTests THEN
	IF NOT bInitDone THEN
		bInitDone := TRUE;
		fbDevValve.Init(
			nId := 1,
			nParentId := 0,
			eResetState := E_ValveResetState.Res_Idle,
			eSafeState := E_ValveResetState.Res_Idle
		);
	END_IF
	
	fbManualController();
	fbDevValve(
		refFbManualCtrl	:= fbManualController,
	);
END_IF

END_PROGRAM

// ---- Axis/FunctionBlocks/Servo/Fb_DevAxisDelta.TcPOU
// Delta ASDA-A2 servo
FUNCTION_BLOCK Fb_DevAxisDelta EXTENDS Fb_DevAxis
VAR
	fbFormatString : FB_FormatString;
    fbCoERead	: FB_CoERead;
	dwErrorCode	: DWORD; // See ASDA A2-E EtherCAT Interface Servo Drive User Manual, chapter 9.2 Error Code Table
END_VAR

SUPER^();

// Continously check drive error code
fbCoERead(
    NetId          := '', 
    Index          := 16#603F, // ASDA2 Error Code
    SubIndex       := 0, 
    pDstBuf        := ADR(dwErrorCode), 
    BufLen         := SIZEOF(dwErrorCode), 
    Execute        := NOT fbCoERead.Busy,
    Timeout        := T#5S, 
    CompleteAccess := FALSE, 
    Axis           := AxisRef
);

IF (dwErrorCode <> 0)
	AND (dwErrorCode <> 16#9000) // Ignore STO errors (already handled by fbDevAxis)
THEN
	stFault.Active := TRUE;
	stFault.FaultType := E_FaultTypes.CF;
	
	// Custom fault descriptions for some common errors
	IF (dwErrorCode = 16#2310) THEN // AL001
		stFault.Description := 'Motor overcurrent';
	ELSIF (dwErrorCode = 16#7305) THEN // AL011
		stFault.Description := 'Encoder error';
	ELSIF (dwErrorCode = 16#7121) THEN // AL030
		stFault.Description := 'Motor protection error (possible overload)';
	ELSIF (dwErrorCode = 16#3300) THEN // AL031
		stFault.Description := 'U,V,W wiring error';
	ELSE // Not so common error
		fbFormatString(sFormat := 'Delta ASDA-A2 servo error: 0x%X', arg1 := F_DWORD(dwErrorCode), sOut => stFault.Description);
	END_IF
END_IF

METHOD INTERNAL ExecReset : BOOL
IF AxisRef.Status.Coupled THEN 
	bResetDone 	:= NOT AxisRef.Status.Error;
	bExec_Reset	R= bResetDone  ;
	RETURN;
END_IF

// ===== reset command =====
	bError 		:= AxisRef.Status.Error OR AxisRef.Status.DriveDeviceError; 
	bExec_Reset	R= fbMcReset.Done  ;

// ==== execute reset functions =====
fbMcReset	( 	Execute	:= bExec_Reset,
				Axis	:= AxisRef ); 
				
// ===== Set feedback =====
	bResetDone 	S= fbMcReset.Done  ;
	bResetDone	R= AxisRef.Status.Error ;
	tonResetDone (IN	:= bResetDone);

// ===== reset limitations =====
	bCmdSafeSpeed 	:= FALSE ;

	
// Reset fault handling 
	IF fbMcReset.Error THEN 
		bError					:= TRUE							;
		stFault.Active 			:= TRUE 						;
		stFault.Description		:= CONCAT('Reset Fault ', UDINT_TO_STRING(fbMcReset.ErrorID));
		stFault.FaultType		:= E_FaultTypes.FF				;
	END_IF
END_METHOD

METHOD PUBLIC Init : BOOL
VAR_INPUT
	// Message location data
	nId			: UINT ; // Identification number of object
	nParentId	: UDINT ; // Id of higher level If aplicable (0 = no parent)
	
	// Config Bits
	bIcfCmdVelocityRpm	: BOOL := FALSE ; // input speeds in Rpm
	bIcfEnableForward 	: BOOL := TRUE 	; // Enable forward motion
	bIcfEnableReverse	: BOOL := TRUE 	; // Enable reverse motion
	bIcfAlwaysEnable	: BOOL := FALSE ; // 1 = Axis always enabled, 0 = Axis disabled at Idle 
	bIcfModuloAxis		: BOOL := FALSE ; // Show axis position as modulo
	bIcfSTOPresent		: BOOL := FALSE ; // Axis safe torque off is present
	bIcfNCHomeSensor	: BOOL := FALSE ; // Homing sensor is inverted (NC)	
	// Config Values 
	mcHomingMode 		: MC_HomingMode := MC_HomingMode.MC_DefaultHoming; 
	fSafeOverride		: LREAL := 10	; // Safe velocity override [%]
	nEncTurnoverVal 	: LREAL := 360	; // encoder turnover value 
	tEnableDelay		: time 	:= T#0MS; // Time between axis enable command and motion command execution (0 := no delay active)	
	tDisabledelay		: TIME 	:= T#100MS; // Axis idle time before axis is disabled 
END_VAR
// ====== Calculate device id =====
	bInitOk :=	ExecIdentifyDevice(nId,nParentId, E_ComponentTypes.Axis) AND bInitOk;

// ====== Set manual device type ======
	eDevType := E_Devices.Axis ;	
	
// ===== Configure Axis =====
	// ***** Config Bits *****
		THIS^.bIcfCmdVelocityRpm	:= bIcfCmdVelocityRpm	; // Enable speed inputs in Rpm
		THIS^.bIcfEnableForward 	:= bIcfEnableForward 	; // Enable forward motion
		THIS^.bIcfEnableReverse		:= bIcfEnableReverse	; // Enable reverse motion
		THIS^.bIcfAlwaysEnable		:= bIcfAlwaysEnable		; // Always enable motor and brake if safety is ok
		THIS^.bIcfModuloAxis		:= bIcfModuloAxis		; // show axis position as modulo
		THIS^.bIcfSTOPresent		:= bIcfSTOPresent		; // Axis has safe torque off function
		THIS^.bIcfNCHomeSensor		:= bIcfNCHomeSensor		; // Axis homing sensor is NC	
	// ***** config homing Mode ***** 
 		THIS^.mcHomingMode 			:= mcHomingMode ; // set homing mode
	// ***** Velocity settings *****
		THIS^.fSafeOverride			:= fSafeOverride	; 	
	// ***** Encoder values *****
		THIS^.fEncoderTurnoverValue := nEncTurnoverVal	; // turnover value for encoder = 25.6 mm per rev * 4096 revolutions 
	// ***** Time delay enable off *****
		THIS^.tEnableDelay		:= tEnableDelay	;
		THIS^.tDisableDelay 	:= tDisabledelay ;		
		
// ===== configure parameters =====
	ParHomeOffset.fMinimum 		:= -1E7;
	ParHomeOffset.fMaximum		:= 1E7;
	ParHomeOffset.nNumber 		:= stIdentity.nLocationId + 1;
	ParHomeOffset.sDiscription  := CONCAT( STR1 := stIdentity.sName, STR2 := ' home position offset');
	ParHomeOffset.sName			:= CONCAT( STR1 := stIdentity.sName, STR2 := ' Home position offset');
	ParHomeOffset.sType			:= 'Cpar';
	ParHomeOffset.sUnit			:= 'unit';
	refFbParHandler.CmdAddParameter( refParameter := ParHomeOffset );

// ===== reset axis state indicators ======
	bError 	:= FALSE;

// ====== Set init to done =======
	bInitOk := TRUE;
	Init := bInitOk;
END_METHOD

END_FUNCTION_BLOCK

// ---- Actuators/Cylinder/Functions/Fb_DevCylWithFbk.TcPOU
{attribute 'reflection'}
FUNCTION_BLOCK PUBLIC Fb_DevCylWithFbk EXTENDS FB_DevValve
VAR_INPUT
	bIcfFbkOpenPresent 	: BOOL := FALSE ; // Feedback for cylinder open is present 
	bIcfFbkClosedPresent: BOOL := FALSE ; // Feedback for Cylinder closed is present
	bIcfCheckTooSlow	: BOOL := TRUE 	; // Check if cylinder is moving too slow
	bIcfCheckTooFast	: BOOL := TRUE 	; // Check if cylinder is moving too fast
	nMargin				: LREAL:= 10	; // % of tollerance in move speed 
END_VAR
VAR_OUTPUT
	// ===== Teach function =======
	bCmdCopyTimeParam 	: BOOL	:= FALSE 	;// Cylinder, Command to higher level copy toucht time to parameters
	bFeClosed			: BOOL 	:= FALSE	; // closed sensor falling edge
	bReClosed			: BOOL 	:= FALSE	; // closed sensor rising edge
	bFeOpen				: BOOL 	:= FALSE 	; // Open sensor falling edge
	bReOpen				: BOOL 	:= FALSE 	; // open sensor rising edge 
	bReOpenSlow         : BOOL  := FALSE    ; // rising edge, opening went too slow
	bReOpenFast         : BOOL  := FALSE    ; // rising edge, opening went too fast
	bReCloseSlow        : BOOL  := FALSE    ; // rising edge, closing went too slow
	bReCloseFast        : BOOL  := FALSE    ; // rising edge, closing went too fast
END_VAR
VAR	
	bFcoCalcDone	: BOOL := FALSE ; // Calculate timers done 
	
	stTimesClose	: Udt_TimerBandwith ; // Timer bandwith for cylinder close
	stTimesOpen		: Udt_TimerBandwith	; // Timer bandwitch for cylinder open 
	
	fbSensorClosed	: Fb_DevDigitalInputFunctions ; // Digital sensor function closed detection
	fbSensorOpen	: Fb_DevDigitalInputFunctions ; // Digital sensor function open detection
	
	fbTimerOpen		: TON ; // Timer measuring cylinder open output has been active
	fbTimerClose 	: TON ; // Timer measuring cylinder close output has been active
	fbTimerTeach	: TON ; // Timer for teaching cylinder 

	rtCmdWriteParam	: R_TRIG ; // Write parameter rising edge trigger 
	// Simulation
	fbTimerSimOpen 	: TON 	; 
	fbTimerSimClose	: TON 	; 
END_VAR

// set device type
	IF eDevType = E_Devices.Undefined THEN 
		eDevType := E_Devices.Cylinder ;
	END_IF

// call base function 
	SUPER^();

// check for device init
	IF NOT bInitOk THEN
		RETURN;
	END_IF 

// ====== Check direction of movement =======
	ExecDirection();
	
// ====== Reset movement indicators =======
	bReOpenSlow  := FALSE;
	bReOpenFast  := FALSE;
	bReCloseSlow := FALSE;
	bReCloseFast := FALSE;

// ====== Check movement speed =======
	ExecTimeout();
	
// ====== Calculate timers =======
	CalcTimers();

// Reduce fault level when in manual mode
IF bManual THEN
	stFault.FaultType		:= E_FaultTypes.OW;
ELSE
	stFault.FaultType		:= E_FaultTypes.CF;
END_IF

METHOD PRIVATE CalcTimers : BOOL
VAR
END_VAR
IF stParTimeToClose.fValue = stTimesClose.Nominal AND stParTimeToOpen.fValue = stTimesOpen.Nominal AND bFcoCalcDone THEN 
	RETURN ;
ELSE
	bFcoCalcDone := FALSE ;
END_IF
 
// ====== Calculate close times ======
	stTimesClose.Nominal 	:= stParTimeToClose.fValue ;
	stTimesClose.Maximum 	:= stParTimeToClose.fValue * (1 + (nMargin / 100));
	stTimesClose.Minimal 	:= stParTimeToClose.fValue * (1 - (nMargin / 100));

// ====== Calculate open times ======
	stTimesOpen.Nominal 	:= stParTimeToOpen.fValue ;
	stTimesOpen.Maximum 	:= stParTimeToOpen.fValue * (1 + (nMargin / 100));
	stTimesOpen.Minimal 	:= stParTimeToOpen.fValue * (1 - (nMargin / 100));
	
// ====== Set feedback =======
	bFcoCalcDone := TRUE ;

// ===== send write parameters command ======	
	rtCmdWriteParam(CLK := bFcoCalcDone);
	bCmdCopyTimeParam := rtCmdWriteParam.Q	;
END_METHOD

METHOD PUBLIC CmdSimulate : BOOL
VAR_INPUT
	bFbkReverse		: BOOL := FALSE ; 
	tTimeSimOpen	: TIME := T#1S 	;
	tTimeSimClose	: TIME := T#1S 	;  
END_VAR
// Run timers when cylinder is active 
	fbTimerSimOpen	(IN := q_Open	, PT := tTimeSimOpen);
	fbTimerSimClose	(IN := q_Close	, PT := tTimeSimClose);

// set feedback sensors to simulate
	fbSensorOpen.bCmdSimulate 	:= TRUE ;
	fbSensorClosed.bCmdSimulate := TRUE ;

// set simulated feedback state 
	IF bFbkReverse THEN 
		fbSensorClosed.bSimState:= fbTimerSimOpen.Q 	;
		fbSensorOpen.bSimState	:= fbTimerSimClose.Q 	; 	
	ELSE 
		fbSensorClosed.bSimState:= fbTimerSimClose.Q 	;
		fbSensorOpen.bSimState	:= fbTimerSimOpen.Q 	; 	
	END_IF
END_METHOD

METHOD PUBLIC CmdTeach : BOOL
VAR_INPUT
END_VAR
// ====== turn off time check function until new calculation cycle =======
	bFcoCalcDone := false ;

// ====== teach cylinder from hardware inputs ======
	fbTimerTeach	(PT:= T#60S);
	fbTimerSwitchDir(PT:= T#1S); 
// ====== time cylinder cycles ======
	// ===== Start test loop =====
	IF bFco_Closed AND fbTimerSwitchDir.Q THEN
		bCmdClose 			:= FALSE;
		bCmdOpen 			:= TRUE ;
		fbTimerSwitchDir.IN	:= FALSE; 
		fbTimerTeach.IN 	:= TRUE ;
	ELSIF bFco_Open AND fbTimerSwitchDir.Q THEN
		bCmdClose 			:= TRUE ;
		bCmdOpen 			:= FALSE;
		fbTimerSwitchDir.IN	:= FALSE; 
		fbTimerTeach.IN 	:= TRUE ;
	ELSIF NOT bCmdClose AND NOT bCmdOpen THEN 
		bCmdClose 			:= TRUE ;
		bCmdOpen 			:= FALSE;
		fbTimerTeach.IN 	:= TRUE ;
	END_IF

// ====== start timing ========
	IF bCmdClose AND bFco_Closed THEN 
		IF fbTimerTeach.IN THEN
			stParTimeToClose.fValue 	:= TIME_TO_LREAL(fbTimerTeach.ET);
		END_IF
		fbTimerSwitchDir.IN := TRUE 		;
		fbTimerTeach.IN 	:= FALSE 		;
	ELSIF bCmdOpen AND bFco_Open THEN 
		IF fbTimerTeach.IN THEN
			stParTimeToOpen.fValue		:= TIME_TO_LREAL(fbTimerTeach.ET);
		END_IF
		fbTimerSwitchDir.IN := TRUE 		;
		fbTimerTeach.IN 	:= FALSE 		;
	END_IF
END_METHOD

METHOD PRIVATE ExecDirection : BOOL
VAR_INPUT
END_VAR
// ===== Check direction commands =====
 	IF q_Close AND fbSensorOpen.bReStatus AND NOT q_Open THEN
		stFault.Active			:= TRUE ;
		stFault.Description		:= 'Cylinder opening instead of closing';
		bErrorActive			:= TRUE 								;
	ELSIF q_Open AND fbSensorClosed.bReStatus AND NOT q_close THEN
		stFault.Active			:= TRUE ;
		stFault.Description		:= 'Cylinder closing instead of opening';
		bErrorActive			:= TRUE 								;
	END_IF
END_METHOD

METHOD PROTECTED ExecSetFeedback : BOOL
VAR_INPUT
END_VAR
{warning disable C0371}
// ====== Call sensor close function =======
	IF bIcfFbkClosedPresent THEN 
		fbSensorClosed();
		bFco_Closed := fbSensorClosed.bFcoInputActive ;
		bFeClosed 	:= fbSensorClosed.bFeStatus ;
		bReClosed 	:= fbSensorClosed.bReStatus ;
	ELSE 
		fbTOnClose	(IN 	:= q_Close, PT 	:= LREAL_TO_TIME(stParTimeToClose.fValue))	;
		bFco_Closed := fbTOnClose.Q ;
	END_IF

// ====== Call sensor open function =======
	IF bIcfFbkOpenPresent THEN 
		fbSensorOpen() 	;
		bFco_open 	:= fbSensorOpen.bFcoInputActive ;
		bFeOpen		:= fbSensorOpen.bFeStatus;
		bReOpen		:= fbSensorOpen.bReStatus;
	ELSE 
		FbTOnOpen	(IN 	:= q_Open, PT 	:= LREAL_TO_TIME(stParTimeToOpen.fValue))	;
		bFco_Open := FbTOnOpen.Q ;
	END_IF

{warning restore C0371}
// ====== set outputs =======
	bReady		:= bFco_Closed OR bFco_Open ;
END_METHOD

METHOD PRIVATE ExecTimeout
VAR
	bEnableCheck : BOOL;
END_VAR
bEnableCheck := (bManual OR bEnable OR (bInitOk AND NOT bIsSafe)) AND bFcoCalcDone;

//====== Run timeout checks for cylinder close =======
IF bEnableCheck AND bIcfFbkClosedPresent THEN 
	IF fbSensorClosed.bReStatus THEN 
		IF bIcfCheckTooFast AND (TIME_TO_LREAL(fbTimerClose.ET) < stTimesClose.Minimal) THEN 
			// send message to HMI 
			stFault.Active			:= TRUE 							;
			stFault.Description		:= 'Cylinder closing too fast';
			bErrorActive			:= TRUE 							;
			bReCloseFast			:= TRUE                             ;
		END_IF
	ELSIF bIcfCheckTooSlow AND fbTimerClose.Q THEN
		// send message to HMI 
		stFault.Active			:= TRUE ;
		stFault.Description		:= 'Cylinder closing too slow';
		bErrorActive			:= TRUE 								;
		bReCloseSlow			:= TRUE                             	;
	END_IF
END_IF	

//====== Run timeout checks for cylinder Open =======
IF bEnableCheck AND bIcfFbkOpenPresent THEN 
	IF fbSensorOpen.bReStatus THEN
		IF bIcfCheckTooFast AND (TIME_TO_REAL(fbTimerOpen.ET) < stTimesOpen.Minimal) THEN 
			// send message to HMI 
			stFault.Active			:= TRUE ;
			stFault.Description		:= 'Cylinder opening too fast';
			bErrorActive			:= TRUE 							;
			bReOpenFast 			:= TRUE 							;
		END_IF
	ELSIF bIcfCheckTooSlow AND fbTimerOpen.Q THEN
		// send message to HMI 
		stFault.Active			:= TRUE ;
		stFault.Description		:= 'Cylinder opening too slow';
		bErrorActive			:= TRUE 							;
		bReOpenSlow 			:= TRUE 							;
	END_IF
END_IF	

//======= run timers =======
fbTimerClose(
	IN := bEnableCheck 
		AND q_Close
		AND	(NOT fbSensorClosed.bFcoInputActive),
	PT := LREAL_TO_TIME(stTimesClose.Maximum)
);
fbTimerOpen(
	IN := bEnableCheck
		AND q_Open
		AND (NOT fbSensorOpen.bFcoInputActive),
	PT := LREAL_TO_TIME(stTimesOpen.Maximum)
);
END_METHOD

METHOD PUBLIC Init : BOOL
VAR_INPUT
	// Message location data
	nId			: UINT ; // Identification number of object
	nParentId	: UDINT ; // Id of higher level If aplicable (0 = no parent)
	// Command state
	eResetState		: E_ValveResetState := 0		; // Cylinder reset state variable (default is idle) 
	eSafeState		: E_ValveResetState	:= 0		; // Valve safe state
END_VAR
bFcoCalcDone := FALSE;

// Enable sensor feedback
fbSensorClosed.bEmbedded := TRUE ;
fbSensorClosed.bEnable	:= TRUE ;
fbSensorClosed.Init	(	nId 		:= 0,
						nParentId 	:= stIdentity.nLocationId) ;

fbSensorOpen.bEmbedded := TRUE ;
fbSensorOpen.bEnable	:= TRUE ;
fbSensorOpen.Init	(	nId 		:= 1,
						nParentId 	:= stIdentity.nLocationId) ;

// Call feedback sensors 
ExecSetFeedback(); 

SUPER^.Init(nId, nParentId, eResetState, eSafeState);

// ===== Set device type for manual control =====
eDevType := E_Devices.Cylinder ;

bInitOk := fbSensorClosed.bInitOk 	AND bInitOk ;
bInitOk := fbSensorOpen.bInitOk		AND bInitOk ;
Init 	:= bInitOk ;
END_METHOD

END_FUNCTION_BLOCK

// ---- Sensors/DigitalSensor/FunctionBlocks/Fb_DevDigitalInputFunctions.TcPOU
{attribute 'reflection'}
FUNCTION_BLOCK PUBLIC Fb_DevDigitalInputFunctions EXTENDS Fb_DevDigitalInput
VAR_OUTPUT
	bFcoDelay			: BOOL			;// Digital sensor, Delayed input status (3 seconds) 
	bFeStatus			: BOOL			;// Digital sensor, Falling edge of input signal	
	bReStatus			: BOOL			;// Digital sensor, Rising edge of input signal
	bFcoFlipFlop		: BOOL			;// Digital sensor, feedback flip flop
	TetInputActive		: TIME			;// Digital sensor, Time elapsed while button is active
END_VAR
VAR
	// ***** Fucntion blocks *****
		FB_delIStatus	: TON	; // Timer function for delayed input status 
		FB_feIStatus	: F_TRIG; // generate falling edge pulse edge from Istatus
		FB_reIStatus	: R_TRIG; // generate falling edge pulse edge from Istatus
		FB_rsIStatus	: RS	; // Set Reset function for flip flop input
END_VAR

SUPER^();


// ====== process functions if enabled ======
	// ***** Set Delayed inputs and time elapsed ****
		FB_delIStatus(	IN:= bFcoInputActive,
						PT:= tDelay , 
						Q=> bFcoDelay , 
						ET=> TetInputActive 
					  ); // Generate delayed input status from push button input status
	// ***** Edge triggers *****
		FB_feIStatus(CLK:= bFcoInputActive , Q=> bFeStatus ); // generate falling edge pulse on pushbutton input
		FB_reIStatus (Clk := bFcoInputActive , Q => bReStatus); // Generate rising edge from push button input signal
	// ***** Flip Flop *****
		FB_rsIStatus(	SET:= bFeStatus AND NOT bFcoFlipFlop , 
						RESET1:= bFeStatus AND bFcoFlipFlop , 
						Q1=> bFcoFlipFlop 
					 ); // Generate set reset function from pushbutton input status

END_FUNCTION_BLOCK

// ---- Sensors/DigitalSensor/FunctionBlocks/Fb_DevDigitalInput.TcPOU
{attribute 'reflection'}
FUNCTION_BLOCK PUBLIC Fb_DevDigitalInput EXTENDS FB_DevBase 
VAR_INPUT
	tDelay				: TIME 	:= T#1S	;// Time before delayed signal becomes active 
	bCmdSimulate		: BOOL 	:= FALSE ;// Simulate sensor Input 
	bSimState			: BOOL 	:= FALSE ;// Simulated sensor state
	bIcfNormalyClosed	: BOOL  := FALSE ;// Hardware input is a normally closed contact
	ibSoftInput			: BOOL 			;// Software input (bFcoInputActive := 
END_VAR
VAR_OUTPUT
	bFcoInputActive		: BOOL 			;// Digital sensor, Button active state
END_VAR
VAR
	Istatus		AT 	%I* : BOOL			;// Digital sensor, Direct input status
END_VAR

// Set device type
IF eDevType = E_Devices.Undefined THEN 
	eDevType := E_Devices.DigitalSensor ;
END_IF

// Call base function
SUPER^();

// ***** Direct input when enabled *****
IF bEnable OR bCmdManual THEN 
	IF bCmdSimulate  THEN 
		bFcoInputActive := bSimState ;
		bCmdSimulate	:= FALSE ;  
	ELSIF bIcfNormalyClosed THEN
		bFcoInputActive := NOT Istatus OR ibSoftInput;
	ELSE
		bFcoInputActive := Istatus OR ibSoftInput ;
	END_IF
ELSE 
	bFcoInputActive := FALSE ;
END_IF

METHOD PUBLIC Init : BOOL
VAR_INPUT
	// Location data for messages  
	nId			: UINT ; // Identification number of object
	nParentId	: UDINT ; // Id of higher level If aplicable (0 = no parent)
END_VAR
// ====== Set init to true =====
	bInitOk	:= TRUE ; 

// ====== Calculate device id =====
	bInitOk :=	ExecIdentifyDevice(nId,nParentId, E_ComponentTypes.DiInput) AND bInitOk;

	Init	:= true ;
END_METHOD

END_FUNCTION_BLOCK

// ---- Axis/FunctionBlocks/Analog/FB_DevAnalogAxis.TcPOU
FUNCTION_BLOCK PUBLIC FB_DevAnalogAxis EXTENDS FB_DevBase
VAR_INPUT
	stManualCtrl 	: ST_ManualAnalogAxisCtrl ; // Manual control
END_VAR
VAR_OUTPUT
	bDriveOk		: BOOL ; // Drive is ok
	bMovingCW		: BOOL ; // Move CW output is active
	bMovingCCW		: BOOL ; // Move CCW output is active
	fActVelocity	: LREAL; // Command velocity of motor
END_VAR
VAR // internal functions 
	fbVelocity		: FB_DevAnalogOutputScaled 	;
	fbqRun			: FB_DevDigitalOutput		;
	fbqReset		: FB_DevDigitalOutput		;
	fbqReverse		: FB_DevDigitalOutput		;
	fbiEnabled		: Fb_DevDigitalInput		;
END_VAR
VAR // Internal commands
	fCmdVelocity	: LREAL;
	bCmdRunCW 		: BOOL ;
	bCmdRunCCW		: BOOL ;
	bCmdReset		: BOOL ;	 
	bInternalEnable : BOOL ;
END_VAR

SUPER^();

// ===== Check inputs =====
	fbiEnabled( bEmbedded	:= TRUE);

IF bInitOk THEN 
	ExecSetOutputs() ;
	bDriveOk	:= fbiEnabled.bFcoInputActive ;
END_IF

METHOD PUBLIC CmdManual : BOOL
VAR_INPUT
END_VAR
bCmdManual := TRUE ;

// Execute Manual commands
	IF stManualCtrl.bCmdRunCW THEN 
		CmdRunCW(fCmdVelocity := stManualCtrl.fCmdVelocity);
	ELSIF stManualCtrl.bCmdRunCCW THEN 
		CmdRunCCW(fCmdVelocity := stManualCtrl.fCmdVelocity);
	END_IF
END_METHOD

METHOD PUBLIC CmdReset : BOOL
VAR_INPUT
END_VAR
bErrorActive 	:= FALSE;

bCmdReset		:= TRUE ;

CmdReset		:= TRUE ;
END_METHOD

METHOD PUBLIC CmdRunCCW : BOOL
VAR_INPUT
	fCmdVelocity	: LREAL ; // Command velocity
END_VAR
bCmdRunCCW			:= TRUE ;
THIS^.fCmdVelocity 	:= fCmdVelocity ; 

CmdRunCCW 	:= bMovingCW ;
END_METHOD

METHOD PUBLIC CmdRunCW : BOOL
VAR_INPUT
	fCmdVelocity	: LREAL ; // Command velocity
END_VAR
bCmdRunCW := TRUE ;
THIS^.fCmdVelocity 	:= fCmdVelocity ;

CmdRunCW 	:= bMovingCW ;
END_METHOD

METHOD PUBLIC CmdSafeStop : BOOL
VAR_INPUT
END_VAR
bIsSafe := TRUE ;

bIsSafe := fbVelocity.CmdSafeStop() AND bIsSafe ;
bIsSafe := fbqRun.CmdSafeStop() 	AND bIsSafe ;
bIsSafe := fbqReverse.CmdSafeStop() AND bIsSafe ;
bIsSafe := fbqReset.CmdSafeStop() 	AND bIsSafe ;

CmdSafeStop := bIsSafe;
END_METHOD

METHOD PRIVATE ExecSetOutputs : BOOL
VAR_INPUT
END_VAR
// ====== Check safety and enable ======
IF fbiEnabled.bFcoInputActive 
AND (bEnable OR bManual) THEN 
	bInternalEnable := TRUE;
ELSE
	fCmdVelocity 	:= 0;
	bCmdRunCW		:= FALSE;
	bCmdRunCCW		:= FALSE;
END_IF 

// ====== Set outputs =======
	fbVelocity	(	bEmbedded 	:= TRUE,
					bEnable		:= bInternalEnable,
					fCmdValue	:= fCmdVelocity);
				
	fbqRun		(	bEmbedded 	:= TRUE,
					bEnable		:= bInternalEnable,
					bCmdOn		:= bCmdRunCW OR bCmdRunCCW);
				
	fbqReverse	(	bEmbedded 	:= TRUE,
					bEnable		:= bInternalEnable,
					bCmdOn		:= bCmdRunCCW);

	fbqReset	(	bEmbedded 	:= TRUE,
					bEnable		:= bInternalEnable,
					bCmdOn		:= bCmdReset);

// ===== reset input commands =====
	fCmdVelocity 	:= 0;
	bCmdRunCW		:= FALSE;
	bCmdRunCCW		:= FALSE;
	bCmdManual		:= FALSE;
	bCmdReset		:= FALSE;
	bInternalEnable := FALSE;
// ===== set feedback =====

bMovingCW		:= fbqRun.bOutputState AND NOT fbqReverse.bOutputState;
bMovingCCW		:= fbqRun.bOutputState AND fbqReverse.bOutputState;
fActVelocity	:= fbVelocity.fOutputValue ;
END_METHOD

METHOD Init : BOOL
VAR_INPUT
	// Message location data
	nId			: UINT ; // Identification number of object
	nParentId	: UDINT ; // Id of higher level If aplicable (0 = no parent)

	// Motor settings
	fMaxVelocity : LREAL ; // Maximum motor velocity for scaling
END_VAR
// ====== initialize components =====
	bInitOk := TRUE ;

// ====== Calculate device id =====
	bInitOk :=	ExecIdentifyDevice(nId, nParentId, E_ComponentTypes.Axis) AND bInitOk;

// ====== Set manual device type ======
	eDevType := E_Devices.AnalogAxis ;	


bInitOk := 	fbVelocity.Init	( 	nId 			:= 0,
								nParentId		:= stIdentity.nLocationId,
								benableNegative	:= FALSE )
								AND bInitOk;
			fbVelocity.SetScaling	(fMaxValue 		:= fMaxVelocity);
								
bInitOk	:= 	fbqRun.Init		( 	nId				:= 1,
								nParentId		:= stIdentity.nLocationId)
								AND bInitOk;

bInitOk	:= 	fbqReset.Init	( 	nId				:= 2,
								nParentId		:= stIdentity.nLocationId)
								AND bInitOk;

bInitOk	:= 	fbqReverse.Init	( 	nId				:= 3,
								nParentId		:= stIdentity.nLocationId)
								AND bInitOk;

bInitOk	:= 	fbiEnabled.Init	( 	nId				:= 4,
								nParentId		:= stIdentity.nLocationId)
								AND bInitOk;

// ====== Set feedback =======
Init := bInitOk;
END_METHOD

END_FUNCTION_BLOCK

// ---- Outputs/AnalogOutputs/FB_DevAnalogOutputScaled.TcPOU
{attribute 'reflection'}
FUNCTION_BLOCK FB_DevAnalogOutputScaled EXTENDS FB_DevAnalogOutput
VAR_INPUT
END_VAR
VAR_OUTPUT
END_VAR
VAR
	fGainFactor 	: LREAL:= 32767	;
END_VAR

SUPER^();

METHOD INTERNAL ExecSetFeedback : BOOL
VAR_INPUT
END_VAR
// Set feedback 
fOutputValue := qnHwOut ;
END_METHOD

METHOD INTERNAL ExecSetOutput : BOOL
VAR_INPUT
END_VAR
// Set Output to physical device
IF (bEnable OR bCmdManual) THEN 
	qnHwOut := LREAL_TO_INT(fCmdValue * fGainFactor) ;
	qnHwOut := LIMIT(nLimitMin, qnHwOut, nLimitMax) ; 
ELSE 
	qnHwOut		:= 0;
	fCmdValue 	:= 0 ; 
END_IF
END_METHOD

METHOD PUBLIC SetScaling : BOOL 
VAR_INPUT
	fMaxValue	: LREAL ; 		// Maximum input value after scaling, e.g. 100% (mandatory input)  
END_VAR
// calculate gain 
fGainFactor := nLimitMax / fMaxValue ;
END_METHOD

END_FUNCTION_BLOCK

// ---- Outputs/AnalogOutputs/FB_DevAnalogOutput.TcPOU
{attribute 'reflection'}
FUNCTION_BLOCK PUBLIC FB_DevAnalogOutput EXTENDS FB_DevBase 
VAR_INPUT
	fCmdValue		: LREAL := 0 ;
END_VAR
VAR_OUTPUT
	fOutputValue	: LREAL := 0 ;
END_VAR
VAR
	nLimitMin		: INT := -32767 ;
	nLimitMax 		: INT := 32767 ;
	qnHwOut	AT%Q*	: INT := 0 ;
END_VAR

// set device type
IF eDevType = E_Devices.Undefined THEN 
	eDevType := E_Devices.AnalogOut ;
END_IF

// Call base function
SUPER^();


// Call private functions
ExecSetOutput();
ExecSetFeedback();

METHOD INTERNAL ExecSetFeedback : BOOL
VAR_INPUT
END_VAR
// Set feedback 
fOutputValue := INT_TO_LREAL(qnHwOut) ;
END_METHOD

METHOD INTERNAL ExecSetOutput : BOOL
VAR_INPUT
END_VAR
// Set Output to physical device
IF (bEnable OR bCmdManual) THEN 
	qnHwOut := LREAL_TO_INT(fCmdValue) ; 
	qnHwOut := LIMIT(nLimitMin, qnHwOut, nLimitMax) ; 
ELSE 
	qnHwOut 	:= 0;
	fCmdValue 	:= 0 ; 
END_IF
END_METHOD

METHOD PUBLIC Init : BOOL
VAR_INPUT
	// Location data for messages  
	nId				: UINT; // Identification number of object
	nParentId		: UDINT; // Id of higher level If aplicable (0 = no parent)
	benableNegative	: BOOL ; // Enable negative values
END_VAR
// ====== Set init to true =====
	bInitOk	:= TRUE ; 

// ====== Calculate device id =====
	bInitOk :=	ExecIdentifyDevice(nId,nParentId, E_ComponentTypes.AnOutput) AND bInitOk;
	
// ====== set minimum value ========
	IF benableNegative THEN 
		nLimitMin := -32767;
	ELSE
		nLimitMin := 0 ;
	END_IF
	
// ====== Set feedback ======
	Init 	:= TRUE ;
END_METHOD

END_FUNCTION_BLOCK

// ---- Outputs/DigitalOutputs/FB_DevDigitalOutput.TcPOU
{attribute 'reflection'}
FUNCTION_BLOCK PUBLIC FB_DevDigitalOutput EXTENDS FB_DevBase
VAR_INPUT
	bCmdOn			: BOOL ; // command output status
END_VAR
VAR_OUTPUT
	bOutputState	: BOOL := FALSE ; // State of physical output
END_VAR
VAR
	qbOutput AT%Q* : BOOL ; // Output to physical device
END_VAR

// Call base function
SUPER^();


// Call private functions
ExecSetOutput();
ExecSetFeedback();

METHOD PRIVATE ExecSetFeedback : BOOL
VAR_INPUT
END_VAR
// Set feedback 
bOutputState := qbOutput ;
END_METHOD

METHOD PRIVATE ExecSetOutput : BOOL
VAR_INPUT
END_VAR
// Set Output to physical device
IF (bEnable OR bCmdManual) THEN 
	qbOutput := bCmdOn ; 
ELSE 
	qbOutput S= FALSE ; 
END_IF
END_METHOD

METHOD PUBLIC Init : BOOL
VAR_INPUT
	// Location data for messages  
	nId			: UINT ; // Identification number of object
	nParentId	: UDINT ; // Id of higher level If aplicable (0 = no parent)
END_VAR
// ====== Set init to true =====
	bInitOk	:= TRUE ; 

// ====== Calculate device id =====
	bInitOk :=	ExecIdentifyDevice(nId,nParentId, E_ComponentTypes.DiOutput) AND bInitOk;

// ====== Set feedback =====
	Init := bInitOk;
END_METHOD

END_FUNCTION_BLOCK

// ---- Axis/FunctionBlocks/ServoHybrid/FB_DevBasicACAxis.TcPOU
{attribute 'reflection'}
FUNCTION_BLOCK PUBLIC FB_DevBasicACAxis EXTENDS FB_DevBase
VAR_INPUT
	// ===== General Function input =====
		fCmdAcc			: LREAL := 15000;
		fCmdDecc		: LREAL := 15000; 
	// Manual control reference
		stManualCtrl	: UDT_ManualAxisCtrl ;
END_VAR
VAR_OUTPUT
	bHomed			: BOOL 	:= FALSE; 
	bMoving		: BOOL ; // Axis is moving
	bInPosition : BOOL ; // Axis is in position 
END_VAR
VAR
		AxisRef	: AXIS_REF ; // reference to AC axis
	// ===== HW Config Bits =====
		bIcfCmdVelocityRpm	: BOOL ; // input speeds in Rpm
		bIcfEnableForward 	: BOOL ; // Enable forward motion
 		bIcfEnableReverse	: BOOL ; // Enable reverse motion
		bIcfAlwaysEnable	: BOOL ; // 1 = Axis always enabled, 0 = Axis disabled at Idle 
		bIcfSimulationMode	: BOOL := FALSE ; // Simulation mode is active [default set to False] 
	// ===== Internal motion values ======
		fHomePosition		: LREAL := 0 ; // set position at homing
	// ====== Axis Settings ======
		fMaxVelo		: LREAL := 0 ; // Axis Maximum velocity
		fMaxAcc			: LREAL := 0 ; // Axis Maximum cceleration
		fMaxDec			: LREAL := 0 ; // axis Maxium deceleration 
		
		fSafeVeloLimit	: LREAL	:= 200; // Safe velocity limit 
		tEnableDelay	: TIME 	:= T#150MS	;
		tDisableDelay	: TIME 	:= T#500MS  ;
		
